IF GVL.Error_code=0 AND GVL.eAzErrorcode = 0 AND NOT GVL.bAzCtrlBit7  AND NOT tr AND NOT bfin1 AND NOT bfin2 THEN
	IF GVL.bLocalCtrl=FALSE THEN //远控
		IF sCtrl.iMode <> 1 THEN
			istate:=0;
			icount:=0;
		END_IF
		CASE sCtrl.iMode OF
			MODES.powerOff: // 下电
				IF NOT sStatus.Disabled THEN
					IF sStatus.Moving THEN // 运动中，先停止运动
						GVL.diAzTargetVel := 0;
						bAzCtrlBit8 := TRUE;
					ELSE
						// 写入下电控制字
						GVL.bAzCtrlBit3 := FALSE;
						GVL.bAzCtrlBit0 := FALSE;
						GVL.bAzCtrlBit1 := FALSE;
						GVL.bAzCtrlBit2 := FALSE;
					END_IF
				END_IF
				
				vpid1(rKpbase:=1, rKibase:=0.01, rKpMax:=1, rKiMax:=0.01, rVelThreshold:=10,rTarget:=sCtrl.rPIDCmdPos,rFeedback:=rRealPos,rPosLimPositive:=sCtrl.rSoft_limit_Postive,
							rPosLimNegitive:=sCtrl.rSoft_limit_Negative,
								bPIDEnable:=sCtrl.bPIDEnable,rVelLim:=sCtrl.rVel_Limit,rKpScale:=0.02,rKiScale:=0.005,rElPos:=GVL.rFctPosReal_1-90,
								iThrehold:=sCtrl.rPIDThre,rPIDOutDir=>sCtrl.rPIDCmdVel);
			MODES.powerOn:  // 上电
				IF sStatus.Disabled THEN
					// 目标速度清零
					GVL.diAzTargetVel := 0;
					IF GVL.siAzMode <> 3 THEN // 上电时模式默认为3，速度模式
						GVL.siAzMode := 3;
					END_IF
					IF siAzMode = 3 THEN
						CASE istate OF
							0:
								GVL.bAzCtrlBit1 := TRUE;
								GVL.bAzCtrlBit2 := TRUE;
								icount := icount + 1;
								IF icount = 20 THEN
									icount:=0;
									istate:=1;
								END_IF
							1:
								GVL.bAzCtrlBit0 := TRUE;
								icount := icount + 1;
								IF icount = 20 THEN
									icount:=0;
									istate:=2;
								END_IF
							2:
								GVL.bAzCtrlBit3 := TRUE;
						END_CASE
					END_IF
				ELSE
					IF sStatus.Moving THEN
						GVL.diAzTargetVel := 0;
						bAzCtrlBit8 := TRUE;
					ELSE
						bAzCtrlBit8 := FALSE;
					END_IF
				END_IF
			MODES.positionMode: // 远控指向模式
				IF NOT sStatus.Disabled THEN
					IF sCtrl.bStartAutoTrack THEN
						//自跟踪模式下，由误差电压直接驱动
						VelPID_1(rTarget:=sCtrl.rChanU + rRealPos,
								rFeedback:=rRealPos,
								rPosLimPositive:=sCtrl.rSoft_limit_Postive,
								rPosLimNegative:=sCtrl.rSoft_limit_Negative,
								rVelLim:=sCtrl.rVel_Limit,
								rKp:=1,//自跟踪PI系数3,0.02
								rKi:=0,
								rKd:=0,
								bPIDEnable:=sCtrl.bPIDEnable,
								iThreshold:= -1,
								rPIDOutput=>sCtrl.rPIDCmdVel);							
					ELSE
						//PID计算速度指令
						VelPID_1(rTarget:=sCtrl.rPosCmd,
							rFeedback:=rRealPos,
							rVelLim:=sCtrl.Pos_Vel,
							rPosLimPositive:=sCtrl.rSoft_limit_Postive,
							rPosLimNegative:=sCtrl.rSoft_limit_Negative,
							rKp:=0.6,//程引PI系数低带：1,0.002  高带：3,0.02
							rKi:=0,
							rKd:=0,
							bPIDEnable:=sCtrl.bPIDEnable,
							iThreshold:=sCtrl.rPIDThre,
							rPIDOutput=>sCtrl.rPIDCmdVel);
					END_IF
					GVL.diAzTargetVel := REAL_TO_DINT(sCtrl.rPIDCmdVel * 524288 / 360);
					GVL.diAzTargetAcc := REAL_TO_UDINT(12 * 524288 / 360);   //加速度
					GVL.diAzTargetDec := REAL_TO_UDINT(12 * 524288 / 360);   //减速度
				END_IF
			MODES.velocityMode://手控速度模式-远控模式
				IF NOT sStatus.Disabled THEN
					IF ABS(sCtrl.rVelCmd) <= sCtrl.rVel_Limit THEN
						GVL.diAzTargetVel := REAL_TO_DINT(sCtrl.rVelCmd * 524288 / 360);
					ELSIF sCtrl.rVelCmd > sCtrl.rVel_Limit THEN
						GVL.diAzTargetVel := REAL_TO_DINT(sCtrl.rVel_Limit * 524288 / 360);
					ELSE
						GVL.diAzTargetVel := REAL_TO_DINT(-sCtrl.rVel_Limit * 524288 / 360);
					END_IF
					GVL.diAzTargetAcc := REAL_TO_UDINT(sCtrl.rAcceleration * 524288 / 360);   //加速度
					GVL.diAzTargetDec := REAL_TO_UDINT(sCtrl.rDeceleration * 524288 / 360);   //减速度
				END_IF
			MODES.programBootMode://PID速度模式-正常模式 程引
				IF NOT sStatus.Disabled THEN
					IF sCtrl.bStartAutoTrack THEN
						(*
						//自跟踪模式下，由误差电压直接驱动
						VelPID_3(rTarget:=sCtrl.rChanU + rRealPos,
								rFeedback:=rRealPos,
								rPosLimPositive:=sCtrl.rSoft_limit_Postive,
								rPosLimNegative:=sCtrl.rSoft_limit_Negative,
								rVelLim:=sCtrl.rVel_Limit,
								rKp:=sCtrl.rP_AutoTrack,//自跟踪PI系数3,0.02
								rKi:=sCtrl.rI_AutoTrack,
								rKd:=sCtrl.rD,
								bPIDEnable:=sCtrl.bPIDEnable,
								iThreshold:= -1,
								rPIDOutput=>sCtrl.rPIDCmdVel);
								*)
						vpid1(rKpbase:=Persistentvars.rAzKpBase, rKibase:=Persistentvars.rAzKiBase, rKpMax:=Persistentvars.rAzKpMax, rKiMax:=Persistentvars.rAzKiMax, rVelThreshold:=Persistentvars.rAzThre,rTarget:=sCtrl.rPIDCmdPos,rFeedback:=rRealPos,rPosLimPositive:=sCtrl.rSoft_limit_Postive,
							rPosLimNegitive:=sCtrl.rSoft_limit_Negative,
								bPIDEnable:=sCtrl.bPIDEnable,rVelLim:=sCtrl.rVel_Limit,rKpScale:=Persistentvars.rAzKpscale,rKiScale:=Persistentvars.rAzKiscale,rElPos:=GVL.rFctPosReal_1-90,
								iThrehold:=sCtrl.rPIDThre,rPIDOutDir=>sCtrl.rPIDCmdVel);							
					ELSE
						//PID计算速度指令
						(*
						VelPID_3(rTarget:=sCtrl.rPIDCmdPos,
							rFeedback:=rRealPos,
							rVelLim:=sCtrl.rVel_Limit,
							rPosLimPositive:=sCtrl.rSoft_limit_Postive,
							rPosLimNegative:=sCtrl.rSoft_limit_Negative,
							rKp:=sCtrl.rP,//程引PI系数地带：1,0.002  高带：3,0.02
							rKi:=sCtrl.rI,
							rKd:=sCtrl.rD,
							bPIDEnable:=sCtrl.bPIDEnable,
							iThreshold:=sCtrl.rPIDThre,
							rPIDOutput=>);
							*)
						vpid1(rKpbase:=Persistentvars.rAzKpBase, rKibase:=Persistentvars.rAzKiBase, rKpMax:=Persistentvars.rAzKpMax, rKiMax:=Persistentvars.rAzKiMax, rVelThreshold:=Persistentvars.rAzThre,rTarget:=sCtrl.rPIDCmdPos,rFeedback:=rRealPos,rPosLimPositive:=sCtrl.rSoft_limit_Postive,
							rPosLimNegitive:=sCtrl.rSoft_limit_Negative,
								bPIDEnable:=sCtrl.bPIDEnable,rVelLim:=sCtrl.rVel_Limit,rKpScale:=Persistentvars.rAzKpscale,rKiScale:=Persistentvars.rAzKiscale,rElPos:=GVL.rFctPosReal_1-90,
								iThrehold:=sCtrl.rPIDThre,rPIDOutDir=>sCtrl.rPIDCmdVel);
						
					END_IF
					GVL.diAzTargetVel := REAL_TO_DINT(sCtrl.rPIDCmdVel * 524288 / 360);
					GVL.diAzTargetAcc := REAL_TO_UDINT(sCtrl.rAcceleration * 524288 / 360);   //加速度
					GVL.diAzTargetDec := REAL_TO_UDINT(sCtrl.rDeceleration * 524288 / 360);   //减速度
				END_IF
			MODES.reset://重置
				IF NOT sStatus.Disabled THEN
					IF sStatus.Moving THEN
						GVL.diAzTargetVel := 0;
						bAzCtrlBit8 := TRUE;
					ELSE
						bAzCtrlBit8 := FALSE;
					END_IF
				END_IF
			MODES.halt://待机
				IF NOT sStatus.Disabled THEN
					IF sStatus.Moving THEN
						GVL.diAzTargetVel := 0;
						bAzCtrlBit8 := TRUE;
					ELSE
						bAzCtrlBit8 := FALSE;
					END_IF
				END_IF
			
		END_CASE
	ELSE // 本控
		IF sLocal.iMode <> 1 THEN
			istate:=0;
			icount:=0;
		END_IF
		CASE sLocal.iMode OF
			MODES.powerOff: // 下电
				IF NOT sStatus.Disabled THEN
					IF sStatus.Moving THEN // 运动中，先停止运动
						GVL.diAzTargetVel := 0;
						bAzCtrlBit8 := TRUE;
					ELSE
						// 写入下电控制字
						GVL.bAzCtrlBit3 := FALSE;
						GVL.bAzCtrlBit0 := FALSE;
						GVL.bAzCtrlBit1 := FALSE;
						GVL.bAzCtrlBit2 := FALSE;
					END_IF
				END_IF
			MODES.powerOn:  // 上电
				IF sStatus.Disabled THEN
					// 目标速度清零
					GVL.diAzTargetVel := 0;
					IF GVL.siAzMode <> 3 THEN // 上电时模式默认为3，速度模式
						GVL.siAzMode := 3;
					END_IF
					IF siAzMode = 3 THEN
						CASE istate OF
							0:
								GVL.bAzCtrlBit1 := TRUE;
								GVL.bAzCtrlBit2 := TRUE;
								icount := icount + 1;
								IF icount = 20 THEN
									icount:=0;
									istate:=1;
								END_IF
							1:
								GVL.bAzCtrlBit0 := TRUE;
								icount := icount + 1;
								IF icount = 20 THEN
									icount:=0;
									istate:=2;
								END_IF
							2:
								GVL.bAzCtrlBit3 := TRUE;
						END_CASE
					END_IF
				ELSE
					IF sStatus.Moving THEN
						GVL.diAzTargetVel := 0;
						bAzCtrlBit8 := TRUE;
					ELSE
						bAzCtrlBit8 := FALSE;
					END_IF
				END_IF
			MODES.velocityMode://手控速度模式-本控模式
				IF NOT sStatus.Disabled THEN
					IF ABS(sLocal.rVelCmd) <= sLocal.rVel_Limit THEN
						GVL.diAzTargetVel := REAL_TO_DINT(sLocal.rVelCmd * 524288 / 360);
					ELSIF sLocal.rVelCmd > sLocal.rVel_Limit THEN
						GVL.diAzTargetVel := REAL_TO_DINT(sLocal.rVel_Limit * 524288 / 360);
					ELSE
						GVL.diAzTargetVel := REAL_TO_DINT(-sLocal.rVel_Limit * 524288 / 360);
					END_IF
					GVL.diAzTargetAcc := REAL_TO_UDINT(sLocal.rAcceleration * 524288 / 360);   //加速度
					GVL.diAzTargetDec := REAL_TO_UDINT(sLocal.rDeceleration * 524288 / 360);   //减速度
				END_IF
			MODES.programBootMode://本控位置模式
				IF NOT sStatus.Disabled THEN
					IF NOT sLocal.bPIDEnable THEN
						GVL.diAzTargetVel := 0;							
					ELSE
						IF NOT slocal.bStartAutoTrack THEN
							//PID计算速度指令
							 VelPID_2(rTarget:=sLocal.rPosCmd,
									 rFeedback:=rRealPos,
									 rPosLimPositive:=sLocal.rSoft_limit_Postive,//软限位
									 rPosLimNegative:=sLocal.rSoft_limit_Negative,
									 rKp:=0.6,
									 rKi:=0,
									 rKd:=0,
									 iThreshold:=sLocal.rPIDThre,
									 bPIDEnable:=sLocal.bPIDEnable,
									 rVelLim:=sLocal.Pos_Vel,
									 rPIDOutput=>sLocal.rPIDCmdVel);//普通PID
						ELSE
							//PID计算速度指令
							 VelPID_2(rTarget:=sLocal.rChanU + rRealPos,
								rFeedback:=rRealPos,
								rPosLimPositive:=sLocal.rSoft_limit_Postive,
								rPosLimNegative:=sLocal.rSoft_limit_Negative,
								rVelLim:=sLocal.rVel_Limit,
								rKp:=1,//自跟踪PI系数3,0.02
								rKi:=0,
								rKd:=0,
								bPIDEnable:=sLocal.bPIDEnable,
								iThreshold:= -1,
								rPIDOutput=>sLocal.rPIDCmdVel);//普通PID
						END_IF
						
					END_IF
					GVL.diAzTargetVel := REAL_TO_DINT(sLocal.rPIDCmdVel * 524288 / 360);
					GVL.diAzTargetAcc := REAL_TO_UDINT(12 * 524288 / 360);   //加速度
					GVL.diAzTargetDec := REAL_TO_UDINT(12 * 524288 / 360);   //减速度
				END_IF
			MODES.reset://重置
			// 是否需要
			MODES.halt://待机
				IF NOT sStatus.Disabled THEN
					IF sStatus.Moving THEN
						GVL.diAzTargetVel := 0;
						bAzCtrlBit8 := TRUE;
					ELSE
						bAzCtrlBit8 := FALSE;
					END_IF
				END_IF
			
		END_CASE
	END_IF
ELSIF GVL.Error_code<>0 AND GVL.eAzErrorcode = 0 AND NOT GVL.bAzCtrlBit7  AND NOT tr AND NOT bfin1 AND NOT bfin2 THEN
	// 出现错误，轴停止运动
	GVL.diAzTargetVel := 0;
	bAzCtrlBit8 := TRUE;
	TON_0(IN:=bAzCtrlBit8,PT:=T#1S,Q=>,ET=>);//判断stop0执行是否超时,若超时强制下电（手动复位）
	IF TON_0.Q THEN
		bTick:=TRUE;
	END_IF
	IF bTick AND sStatus.Moving THEN // 超时强制下电
		// 写入下电控制字
		GVL.bAzCtrlBit3 := FALSE;
		GVL.bAzCtrlBit0 := FALSE;
		GVL.bAzCtrlBit1 := FALSE;
		GVL.bAzCtrlBit2 := FALSE;
	END_IF
END_IF

END_FUNCTION_BLOCK

// Device/Application/PID
FUNCTION_BLOCK PID
VAR_INPUT
    rTarget : REAL;       (* 设定值 *)
    rFeedback : REAL;       (* 反馈值 *)
	rPosLimPositive:LREAL;//位置正限位
	rPosLimNegative:LREAL;//位置反限位
	rKp:REAL;     //比例增益
	rKi:REAL;     //积分增益
	rKd:REAL;     //微分增益
	iThreshold:INT;//积分项开启的位置阈值
	bPIDEnable:BOOL:=TRUE;//PID使能
	rVelLim:LREAL;//速度限制
END_VAR
VAR_OUTPUT
    rPIDOutput : LREAL:=0;         //带方向的输出速度
	rPIDtrace : LREAL:=0;         //带方向的输出速度
END_VAR
VAR
	//rPIDOutPut: REAL:=0.0;
	rLastError: LREAL:=0.0;(*上一次误差*)
	rErrorNow:LREAL:=0.0;(*当前误差*)
    rIntegralNew : LREAL := 0.0; (* 积分项 *)
    rDerivativeNew : LREAL := 0.0; (* 微分项 *)
	rDelta: LREAL;(*增量*)
	rProportionNew: LREAL;
	
	//iAzPIDEnable: INT;
END_VAR


IF (bPIDEnable>0) THEN //如果PID使能
	IF rTarget=rFeedback THEN
		rPIDOutput:=0;	
	ELSE
	
		rErrorNow:=rTarget-rFeedback;//计算当前误差 en
		rProportionNew:=rErrorNow;//比例项
		//积分项
		IF rFeedback>rPosLimNegative AND rFeedback<rPosLimPositive THEN //若在软限位之内，工作时开启积分项
			IF (ABS(rTarget-rFeedback)<iThreshold) THEN//位置差小于积分阈值
				rIntegralNew:= rIntegralNew+rErrorNow; //积分项
			ELSE
				rIntegralNew:=0;
			END_IF;
		ELSE //不在软限位范围内,则积分项为0
			rIntegralNew:=0;
		END_IF

		//PID输出
		rPIDOutPut:=rKp*rProportionNew+rKi*rIntegralNew;
		rPIDtrace:=rKp*rProportionNew+rKi*rIntegralNew;


		//PID限速
		
			IF rPIDOutput<(-rVelLim) THEN
				rPIDOutput:=-rVelLim;
			ELSIF rPIDOutput>rVelLim THEN
				rPIDOutput:=rVelLim;
			END_IF
		
		
		IF rFeedback>rPosLimPositive AND rPIDOutput>0 THEN 
			rPIDOutput:=0;
		END_IF
		IF rFeedback<rPosLimNegative AND rPIDOutput<0 THEN
			rPIDOutput:=0;
		END_IF
		
		rLastError:=rErrorNow;//将当前误差赋值给上一次误差
		
	END_IF
ELSE//非使能清零PID各项
	rProportionNew:=0.0;
	rIntegralNew:=0.0;
	rPIDOutput:=0.0;
END_IF

END_FUNCTION_BLOCK

// Device/Application/vpid
FUNCTION_BLOCK vpid
VAR_INPUT
	rTarget : REAL;           // 设定值
    rFeedback : REAL;         // 反馈值
    rPosLimPositive : LREAL;  // 位置正限位
    rPosLimNegitive : LREAL;  // 位置反限位
    rKpBase : REAL;           // 基础比例增益
    rKiBase : REAL;           // 基础积分增益
    rVelThreshold : LREAL;     // 速度阈值，真实值除以控制频率
    rKpScale : REAL;          // 比例增益比例因子
    rKiScale : REAL;          // 积分增益比例因子
    iThrehold : INT;          // 积分项开启的位置阈值
    bPIDEnable : BOOL := TRUE;// PID使能
    rVelLim : LREAL;          // 速度限制
	rKpMax : REAL;
	rKiMax : REAL;
	rElPos : REAL;            // 俯仰角度
END_VAR

VAR_OUTPUT
    rPIDOutput : LREAL := 0;  // 控制量
	rPIDOutDir: LREAL;
END_VAR

VAR
    rLastFeedback : LREAL := 0.0; // 上一次反馈值
    rErrorNow : LREAL := 0.0;     // 当前误差
    rIntegralNew : LREAL := 0.0;  // 积分项
    rDelta : LREAL;               // 增量
    rProportionNew : LREAL;       // 比例项
    rSpeed : REAL;                // 当前速度
    rKp : REAL:=1;                   // 动态比例增益
    rKi : REAL:=0.02;                   // 动态积分增益
	rInterValueNow : LREAL := 0.0;        // 当前插值位置
	rInterValueLast : LREAL := 0.0;       // 上一次插值位置
	//rSlope :LREAL :=0; 			  //PI变化斜率
	rStep:LREAL:=0.002;                //PI变化率
	
	rKpTarget :REAL:=1;
	rKiTarget :REAL:=0.02;
	
	
END_VAR

IF (bPIDEnable) THEN // 如果PID使能
    IF rTarget = rFeedback THEN
        rPIDOutDir := 0;    
    ELSE
        rErrorNow := rTarget - rFeedback; // 计算当前误差
        rProportionNew := rErrorNow;      // 比例项
		
		IF rElPos > rVelThreshold THEN
			rKpTarget := rKpBase + rKpScale * (rElPos - rVelThreshold);
			rKiTarget := rKiBase + rKiScale * (rElPos - rVelThreshold);
		ELSE
			rKpTarget := rKpBase;
			rKiTarget := rKiBase;
		END_IF
//         rInterValueLast := rInterValueNow; // 将当前插值位置值赋值给上一次
// 		rInterValueNow := RealTimePosCal.ElCubicInter.sout*10000.0;
//         // 计算当前速度
//         // rSpeed := ABS(rFeedback - rLastFeedback);
//         rSpeed := ABS(rInterValueNow - rInterValueLast)/10000.0;
// 		
//         // 根据速度调整PI增益
//         IF rSpeed > rVelThreshold THEN
//             rKpTarget := rKpBase + rKpScale * (rSpeed - rVelThreshold);
//             rKiTarget := rKiBase + rKiScale * (rSpeed - rVelThreshold);
//         ELSE
//             rKpTarget := rKpBase;
//             rKiTarget := rKiBase;
//         END_IF
        IF rKpTarget > rKpMax THEN
			rKpTarget := rKpMax;
		END_IF
		IF rKiTarget > rKiMax THEN
			rKiTarget := rKiMax;
		END_IF
		
		IF rKp<=rKpTarget THEN
			rKp:=rKp+rStep;
		ELSE
			rKp:=rKp-rStep;
		END_IF
		IF rKi<=rKiTarget THEN
			rKi:=rKi+(rKiScale/rKpScale)*rStep;
		ELSE
			rKi:=rKi-(rKiScale/rKpScale)*rStep;
		END_IF
	END_IF
        // 积分项
        IF rFeedback > rPosLimNegitive AND rFeedback < rPosLimPositive THEN // 若在软限位之内，工作时开启积分项
            IF (ABS(rTarget - rFeedback) < iThrehold) THEN // 位置差小于积分阈值
                rIntegralNew := rIntegralNew + rErrorNow;  // 积分项
            ELSE
                rIntegralNew := rIntegralNew;  // 积分项
            END_IF;
        ELSE // 不在软限位范围内，则积分项为0
            rIntegralNew := 0;
        END_IF
        (*
        // 防止目标位置与当前位置偏差过大，导致比例项输出太大，引起震动
        IF rKp * rProportionNew > 2 THEN
            rPIDOutput := 2;
        ELSIF rKp * rProportionNew < -2 THEN
            rPIDOutput := -2;
        ELSE
            rPIDOutput := rKp * rProportionNew + rKi * rIntegralNew / 1000.0; // 由于需求积分项过小，因此积分系数在接口数据上除1000
        END_IF
        *)
		rPIDOutput := rKp * rProportionNew + rKi * rIntegralNew; // 由于需求积分项过小，因此积分系数在接口数据上除1000
        // 根据方向设置输出
        IF rPIDOutput < 0 THEN

            rPIDOutDir := rPIDOutput;
        ELSE

            rPIDOutDir := rPIDOutput;
        END_IF
        
        // PID限速
        IF (ABS(rPIDOutDir) > rVelLim) THEN
            IF rPIDOutDir < (-rVelLim) THEN
                rPIDOutDir := -rVelLim;
            ELSIF rPIDOutDir > rVelLim THEN
                rPIDOutDir := rVelLim;
            END_IF
        END_IF
        
        // 位置限位检查
        IF rFeedback > rPosLimPositive AND rPIDOutDir > 0  THEN
            rPIDOutDir := 0;
        END_IF
        IF rFeedback < rPosLimNegitive AND rPIDOutDir <= 0 THEN
            rPIDOutDir := 0;
        END_IF
        
        //rLastFeedback := rFeedback; // 将当前反馈值赋值给上一次反馈值
		//rInterValueLast := rInterValueNow; // 将当前插值位置值赋值给上一次

ELSE // 非使能清零PID各项
    rProportionNew := 0.0;
    rIntegralNew := 0.0;
    rPIDOutDir := 0.0;
    rPIDOutput := 0.0;
END_IF

END_FUNCTION_BLOCK

// Device/Application/扫描搜索/AGCMaxSearch_PB_1
FUNCTION_BLOCK AGCMaxSearch_PB_1 //双轴静止星步进跟踪使用的代码
VAR_INPUT
	bstart:BOOL;//模块开始标识
	rAGCNow:REAL;//当前AGC值
	btrig:BOOL;//触发一次
	rStepBiasNow:REAL;//当前拉偏量 //用来判断此次搜索是否有效
	bAutoTracking:BOOL;// 自跟踪标识
	bStop:BOOL;//满足ua ue很小
	
	rCurrentPos:REAL;//当前位置
	rInterPos:REAL;//插值位置
	//rOutStepBias:REAL;//外部拉偏量
END_VAR
VAR_OUTPUT
	
	rAGCMaxBias:REAL;//输出AGC最强时的拉偏量 单位为°
	bSucess :BOOL;//数出模块是否成功
	rStepBias:REAL;//步进量
END_VAR
VAR
	ton:Standard.TON;
	rTrg:Standard.R_TRIG;//初始化上升沿检测器
	rAGCInit:REAL:=0;//初始化AGC
	rPrevAGC:REAL:=0;//上一步的AGC值 单位为V
	rBiasInit:REAL;//初始化拉偏量
	
	iCountStep:INT:=0;//计步数
	toN1: Standard.Ton;//计时器 定时触发上升沿 
	
	rDirection: INT:=1;
	rSearchNextStepTarget:REAL;//搜索当前目标位置 单位为°
	rStep:REAL:=0.0003;//步进值
	rSensitivity:REAL:=0.05;//反向灵敏度
	iCountStopMax:INT:=20;//停止计数上限
	
	rLastDirection:INT;//上一次方向，判断是否换向
	iCountDirChange:INT;//换向标识
	rAGCMaxPos:REAL;//信号最强位置
	
	rAGCLastrecord: REAL;
	iStatus: INT;
	iCountStop1:INT;//第一阶段停止标识 (正向)
	iCountStop2:INT;//(反向)
	
	rAGCMaxValue: REAL;//AGC最大值
	
	//新加的
	iCountSearchRight:INT;//搜索方向正确，提前结束标识
	
	bSearchRight:BOOL;//搜索正确标识
	//模块指行完成标识
	iCountBlockEnd:INT;//用来计数确认已达到最强位置
	iCountBlockEndMax:INT:=500;//到位计数上限
END_VAR


rTrg(CLK:=bstart,Q=>);

IF rTrg.Q THEN
	rAGCInit:=rAGCNow;
	rAGCMaxValue:=rAGCNow;
	//rBiasInit:=rCurrentPos-rInterPos;//获取启动时的拉偏量
END_IF

IF bstart THEN
	//搜索换向两次
	IF iCountDirChange=2 THEN
		rSearchNextStepTarget:=rAGCMaxBias;
		IF rStepBias< rSearchNextStepTarget THEN 
			rStepBias:=rStepBias+rStep;
		ELSIF rStepBias> rSearchNextStepTarget THEN
			rStepBias:=rStepBias-rStep;
		ELSE
			rStepBias:=rStepBias;
		END_IF
		
		IF ABS((rInterPos+rStepBias)-rCurrentPos)<0.002 THEN //若位置达到最强位置，则输出成功 //可能只是路过这里,需要持续
			//需要判断稳定
			iCountBlockEnd:=iCountBlockEnd+1;
		ELSE
			iCountBlockEnd:=0;
		END_IF
		IF iCountBlockEnd>iCountBlockEndMax THEN
			iCountBlockEnd:=iCountBlockEndMax+1;
			//用TON1秒后触发
			ton(IN:=TRUE,PT:=T#1S,Q=>,ET=>);
		END_IF
		IF ton.Q THEN
			bSucess:=TRUE;
		END_IF
	ELSE
		rStepBias:=rStepBias+rDirection*rStep;
		IF rDirection<0 THEN
			//若是向小走
			IF rCurrentPos<rInterPos THEN
				IF rAGCNow<rAGCMaxValue-rSensitivity THEN
					iCountStop1:=iCountStop1+1;
					IF iCountStop1>iCountStopMax THEN
						iCountStop1:=iCountStopMax+1;
						IF bSearchRight THEN
							iCountDirChange:=2;
						ELSE
							iCountDirChange:=iCountDirChange+1;
						END_IF
						rDirection:=rDirection*(-1);
					END_IF
				ELSE
					iCountStop1:=0;	
				END_IF
				
				//新加的 测试第一阶段搜索正确后不进行第二次搜索
				IF rAGCNow>rAGCInit+rSensitivity THEN
					iCountSearchRight:=iCountSearchRight+1;
				ELSE
					iCountSearchRight:=0;
				END_IF
				IF iCountSearchRight>200 THEN
					iCountSearchRight:=201;
					bSearchRight:=TRUE;
				END_IF
				
			END_IF
		ELSE
			//若是向正走
			IF rCurrentPos>rInterPos THEN
				IF rAGCNow<rAGCMaxValue-rSensitivity THEN
					iCountStop2:=iCountStop2+1;
					IF iCountStop2>iCountStopMax THEN
						iCountStop2:=iCountStopMax+1;
						IF bSearchRight THEN
							iCountDirChange:=2;
						ELSE
							iCountDirChange:=iCountDirChange+1;
						END_IF
						rDirection:=rDirection*(-1);
					END_IF
				ELSE
					iCountStop2:=0;	
				END_IF
				
				//新加的
				IF rAGCNow>rAGCInit+rSensitivity THEN
					iCountSearchRight:=iCountSearchRight+1;
				ELSE
					iCountSearchRight:=0;
				END_IF
				IF iCountSearchRight>200 THEN
					iCountSearchRight:=201;
					bSearchRight:=TRUE;
				END_IF
				
			END_IF
		END_IF
		(*
		IF rAGCNow<rAGCInit-0.05 THEN
			iCountStop1:=iCountStop1+1;
			IF iCountStop1>150 THEN
				iCountDirChange:=iCountDirChange+1;
				rDirection:=rDirection*(-1);
			END_IF
		ELSE
			iCountStop1:=0;	
		END_IF
		*)
		
		 // 记录最强信号的拉偏量和值
		//IF rAGCNow >= rAGCInit AND rAGCNow> rAGCMaxValue THEN
		IF  rAGCNow> rAGCMaxValue THEN
			rAGCMaxBias := rStepBias;
			rAGCMaxValue := rAGCNow;
		END_IF
	END_IF
ELSE
	rStepBias:=0;
	//清空变量
	iCountDirChange:=0;
	rAGCInit:=0;
	rAGCMaxValue:=0;
	rAGCMaxBias:=0;
	rDirection:=1;
	iCountStop1:=0;
	iCountStop2:=0;
	ton(IN:=FALSE,PT:=T#1S,Q=>,ET=>);
	//rStepBias:=0;
	rSearchNextStepTarget:=0;
	bSucess:=FALSE;
	iCountSearchRight:=0;
	bSearchRight:=FALSE;
	iCountBlockEnd:=0;
END_IF


(*
IF rStepBias< rSearchNextStepTarget THEN 
	rStepBias:=rStepBias+rStep;
ELSIF rStepBias> rSearchNextStepTarget THEN
	rStepBias:=rStepBias-rStep;
ELSE
	rStepBias:=rStepBias;
END_IF*)

END_FUNCTION_BLOCK

// Device/Application/El_ctrl_1
PROGRAM El_ctrl_1
VAR
    Axis1_Ctrl : El_Ctrl_FB;
    bRemote2LocalStop : BOOL;
    bLocal2RemoteStop : BOOL;
    Error : INT;
    Axis1Limit_pos : REAL;
    Axis1Limit_Neg : REAL;
    bRTriger : Standard.R_TRIG;
    bFTriger : Standard.F_TRIG;
    Stop1_Count : INT;
    bStop_1 : BOOL;
    rPosModeStepBias : LREAL;
    rPosModeStep : LREAL := 0.005;
    rStepBiasMax : LREAL := 2;
    rStepBias : LREAL;
    rStep : LREAL := 0.002;
    rAuToStepBias : LREAL;
    rAuToStepBiasTemp : LREAL;
    rAutoStep : LREAL := 0.01;
    TbAutoTrigger : Standard.F_TRIG;
    RbAutoTrigger : Standard.R_TRIG;
    rAutoTrackingBiasMax : LREAL := 6;
    rLocalInitPosModeSpeed : REAL;
    rRemoteInitPosModeSpeed : REAL;
    iCountOffAuto : INT;
    iCasePBAutoTrack : INT := 2;
    rKAuToStepBias : LREAL := 0.45; // 对齐2.4
    agcmaxsearch_tb : AGCMaxSearch_PB_1;
    rSearchNextStepTarget_tb : REAL;
    agcmaxsearch_pb : AGCMaxSearch_PB_1;
    rElthreshold : REAL := 4.2;
    toN1 : Standard.Ton;
    ttime1 : TIME := T#200mS;
    bstartagcmaxsearch : BOOL;
    rSearchNextStepTarget : REAL;
    rMaxPosTest : REAL;
END_VAR

(*
//远控轴参量赋值
Axis1Remote.iMode:=Modbus_Slave.iMode_1;
Axis1Remote.rVelCmd:=Modbus_Slave.rVelcmd_1;
Axis1Remote.rPosCmd:=Modbus_Slave.rPosCmd_1;
Axis1Remote.rP:=Modbus_Slave.rP_1;
Axis1Remote.rI:=Modbus_Slave.rI_1;
Axis1Remote.rD:=Modbus_Slave.rD_1;
Axis1Remote.rPIDThre:=Modbus_Slave.rThreshold_1;
Axis1Remote.rAcceleration:=Modbus_Slave.rAcceleration_1;
Axis1Remote.rDeceleration:=Modbus_Slave.rDeceleration_1;
Axis1Remote.rVel_Limit:=Modbus_Slave.rVelLim_1;
*)
// 方位状态写入
Axis1Status.Error := GVL.bElStsBit3;
Axis1Status.ErrorID := GVL.eElErrorcode;
Axis1Status.bServo_Enable := GVL.bElStsBit0 AND GVL.bElStsBit1 AND GVL.bElStsBit2;
Axis1Status.bBrake := NOT (GVL.bElStsBit0 AND GVL.bElStsBit1 AND GVL.bElStsBit2);
Axis1Status.Disabled := NOT (GVL.bElStsBit0 AND GVL.bElStsBit1 AND GVL.bElStsBit2);
Axis1Remote.rSoft_limit_Negative:=93;Axis1Remote.rSoft_limit_Postive:=180;
Axis1Local.rSoft_limit_Negative:=93;Axis1Local.rSoft_limit_Postive:=180;

//速度的写入
rFctVelReal_1:=DINT_TO_REAL(diElActVel)/524288.0*360.0;
//位置的写入，方位0对应编码器0，所以实际方位是：-1*编码器值
//rFctPosReal_1:=DINT_TO_REAL(diElActPos)/524288.0*360.0 + 5.339;
rFctPosReal_1:=DINT_TO_REAL(diElActPos)/524288.0*360.0 + modbus_slave.lrElOffset;
//软限位控制
Axis1Limit_pos:=180;
Axis1Limit_Neg:=93;
IF Axis1Remote.rPosCmd>Axis1Limit_pos THEN
	Axis1Remote.rPosCmd:=180;
ELSIF Axis1Remote.rPosCmd<Axis1Limit_Neg THEN
	 Axis1Remote.rPosCmd:=93;  
END_IF

IF Axis1Local.rPosCmd>Axis1Limit_pos THEN
	Axis1Local.rPosCmd:=180;
ELSIF Axis1Local.rPosCmd<Axis1Limit_Neg THEN
	 Axis1Local.rPosCmd:=93;  
END_IF

//停止标志符号判断
IF  ABS(rFctVelReal_1)<0.035 THEN
	Stop1_Count:=Stop1_Count+1;
	IF Stop1_Count>100 THEN
		Stop1_Count:=101;
		bStop_1:=TRUE;;
	END_IF
ELSE
	Stop1_Count:=0;
	bStop_1:=FALSE;
END_IF
Axis1Status.Moving := NOT bStop_1;
//PID使能赋值
IF Axis1Remote.iMode=2 OR Axis1Remote.iMode=4 THEN
	Axis1Remote.bPIDEnable:=TRUE;
ELSE
	Axis1Remote.bPIDEnable:=FALSE;
END_IF

//本远控逻辑保护
//远控切本控逻辑保护
bRTriger(CLK:=GVL.bLocalCtrl);
bFTriger(CLK:=GVL.bLocalCtrl);

IF Axis1Status.bServo_Enable AND (bRTriger.Q ) THEN//如果速度不为0且本控发生切换，则减速停止标识为True
	bRemote2LocalStop:=TRUE;
END_IF
IF bRemote2LocalStop  THEN //若减速停止标识符为True 
	
	IF  bStop_1=TRUE THEN//且电机速度不为0 开始减速 减速完成后下使能，下使能完成后复位标识符复位
		Axis1Local.iMode:=0;
		Axis1Remote.iMode:=0;
		IF Axis1Status.bServo_Enable=FALSE THEN
			bRemote2LocalStop:=FALSE;
		END_IF
	ELSE
		Axis1Local.iMode:=7;
		Axis1Remote.iMode:=7;
	END_IF
END_IF

//本控切远控
IF Axis1Status.bServo_Enable AND (bFTriger.Q ) THEN//如果速度不为0且本控发生切换，则减速停止标识为True
	bLocal2RemoteStop:=TRUE;
END_IF
IF bLocal2RemoteStop  THEN //若减速停止标识符为True 
	
	IF  bStop_1=TRUE THEN//且电机速度不为0 开始减速 减速完成后下使能，下使能完成后复位标识符复位
		Axis1Local.iMode:=0;
		Axis1Remote.iMode:=0;
		IF Axis1Status.bServo_Enable=FALSE THEN
			bLocal2RemoteStop:=FALSE;
		END_IF
	ELSE
		Axis1Remote.iMode:=7;
		Axis1Local.iMode:=7;
	END_IF
END_IF
(*
//自跟踪
IF GVL.bStartTrack THEN
	Axis1Remote.bStartAutoTrack := TRUE;
	Axis1Remote.rChanU := AutoTrackingCal.rChanUe;
ELSE
	Axis1Remote.bStartAutoTrack := FALSE;	
	Axis1Remote.rChanU := 0;
END_IF
*)
IF Axis1Remote.iMode=2 THEN
			IF GVL.Chan1AGC>=(GVL.Chanthreshold-0.1) THEN
					agcmaxsearch_pb(bstart:=Az_ctrl_1.agcmaxsearch_tb.bSucess,rAGCNow:=GVL.Chan1AGC,btrig:=Az_ctrl_1.bstartSearchEl,
						rCurrentPos:=rFctPosReal_1,rInterPos:=Axis1Remote.rPosCmd,
				//rOutStepBias:=rStepBias,	
				rStepBiasNow:=rStepBias,bAutoTracking:=GVL.bStartTrack,bStop:=FALSE,
				rStepBias=>rSearchNextStepTarget_tb,rAGCMaxBias=>rMaxPosTest,bSucess=>);
			ELSE
				bstartagcmaxsearch:=FALSE;
				agcmaxsearch_pb(bstart:=Az_ctrl_1.agcmaxsearch_tb.bSucess,rAGCNow:=GVL.Chan1AGC,btrig:=Az_ctrl_1.bstartSearchEl,
				rCurrentPos:=rFctPosReal_1,rInterPos:=Axis1Remote.rPosCmd,
				//rOutStepBias:=rStepBias,
				rStepBiasNow:=rStepBias,bAutoTracking:=GVL.bStartTrack,bStop:=FALSE,
				rStepBias=>rSearchNextStepTarget_tb,rAGCMaxBias=>rMaxPosTest,bSucess=>);
			END_IF
		ELSIF Axis1Remote.iMode=4 AND rFctPosReal_1-90>rElthreshold  THEN
			IF GVL.Chan1AGC>=(GVL.Chanthreshold-0.1) THEN
					agcmaxsearch_pb(bstart:=Az_ctrl_1.agcmaxsearch_pb.bSucess,rAGCNow:=GVL.Chan1AGC,btrig:=Az_ctrl_1.bstartSearchEl,
						rCurrentPos:=rFctPosReal_1,rInterPos:=RealTimePosCal.rInterElPos,
				//rOutStepBias:=rStepBias,	
				rStepBiasNow:=rStepBias,bAutoTracking:=GVL.bStartTrack,bStop:=FALSE,
				rStepBias=>rSearchNextStepTarget,rAGCMaxBias=>rMaxPosTest,bSucess=>);
			ELSE
				bstartagcmaxsearch:=FALSE;
				agcmaxsearch_pb(bstart:=Az_ctrl_1.agcmaxsearch_pb.bSucess,rAGCNow:=GVL.Chan1AGC,btrig:=Az_ctrl_1.bstartSearchEl,
				rCurrentPos:=rFctPosReal_1,rInterPos:=RealTimePosCal.rInterElPos,
				//rOutStepBias:=rStepBias,
				rStepBiasNow:=rStepBias,bAutoTracking:=GVL.bStartTrack,bStop:=FALSE,
				rStepBias=>rSearchNextStepTarget,rAGCMaxBias=>rMaxPosTest,bSucess=>);
			END_IF
			//把rSearchNextStepTarget附加到AzCtrl.rPIDCmdPos上
		ELSIF Axis1Remote.iMode =0  OR Axis1Remote.iMode =7 THEN
			bstartagcmaxsearch:=FALSE;
			//rSearchNextStepTarget:=0;
			agcmaxsearch_pb(bstart:=Az_ctrl_1.agcmaxsearch_pb.bSucess,rAGCNow:=GVL.Chan1AGC,btrig:=Az_ctrl_1.bstartSearchEl,
			rCurrentPos:=rFctPosReal_1,rInterPos:=RealTimePosCal.rInterElPos,	
			//rOutStepBias:=rStepBias,
			rStepBiasNow:=rStepBias,bAutoTracking:=GVL.bStartTrack,bStop:=FALSE,
			rStepBias=>rSearchNextStepTarget,rAGCMaxBias=>rMaxPosTest,bSucess=>);
		END_IF
// 程引模式下自跟踪拉偏
IF GVL.bStartTrack AND Axis1Remote.iMode=4 THEN
	Axis1Remote.bStartAutoTrack := TRUE;
	IF rAuToStepBias > rAutoTrackingBiasMax THEN
		rAuToStepBias := rAutoTrackingBiasMax;
	ELSIF rAuToStepBias < -rAutoTrackingBiasMax THEN
		rAuToStepBias := -rAutoTrackingBiasMax;
	ELSE
		rAuToStepBiasTemp:=0.02*AutoTrackingCal.rDirSenFac*AutoTrackingCal.rChanUe;
		rAuToStepBias:=rAuToStepBias+AutoTrackingCal.rDirSenFac*rKAuToStepBias*AutoTrackingCal.rChanUe/1000.0;
	END_IF
ELSIF NOT GVL.bStartTrack AND Axis1Remote.iMode=4 THEN
	IF 	rAuToStepBias>0 THEN//关闭自跟踪后自跟踪拉偏量逐渐归0
		rAuToStepBias:=rAuToStepBias-rAutoStep;
	ELSIF rAuToStepBias<0 THEN
		rAuToStepBias:=rAuToStepBias+rAutoStep;
	ELSE
		rAuToStepBias:=0;
	END_IF
	
	IF Modbus_Slave.rBias_1>rStepBias THEN
		rStepBias:=rStepBias+rStep;
		IF rStepBias>=Modbus_Slave.rBias_1 THEN
			rStepBias:=Modbus_Slave.rBias_1;
		END_IF
	ELSIF Modbus_Slave.rBias_1<rStepBias THEN
		rStepBias:=rStepBias-rStep;
		IF rStepBias<=Modbus_Slave.rBias_1 THEN
			rStepBias:=Modbus_Slave.rBias_1;
		END_IF
	END_IF
	rAuToStepBiasTemp:=0;
ELSIF GVL.bStartTrack AND Axis1Remote.iMode=2 THEN
	Axis1Remote.bStartAutoTrack := TRUE;
	Axis1Remote.rChanU := AutoTrackingCal.rChanUe;
ELSE
	Axis1Remote.bStartAutoTrack := FALSE;	
	rAuToStepBias:=0;
	rStepBias:=0;
	rAuToStepBiasTemp:=0;
END_IF

//本控自跟踪
IF GVL.bStartLocalAutoTrack AND Axis1Local.iMode = 4 THEN
	Axis1Local.bStartAutoTrack := TRUE;
	Axis1Local.rChanU := AutoTrackingCal.rChanUeLocal;
ELSE
	Axis1Local.bStartAutoTrack := FALSE;
END_IF

//拉偏
Axis1Remote.rPIDCmdPos:=RealTimePosCal.rInterElPos+rStepBias+rAuToStepBias+rSearchNextStepTarget+SECURITYCHECK.el_out+rAuToStepBiasTemp;
//限位
IF Axis1Remote.rPIDCmdPos<93 THEN
	Axis1Remote.rPIDCmdPos:=93;
ELSIF Axis1Remote.rPIDCmdPos>180 THEN
	Axis1Remote.rPIDCmdPos:=180;
END_IF

Axis1_Ctrl(sLocal:=Axis1Local, sCtrl:=Axis1Remote, sStatus:=Axis1Status, sVisible:=Axis1Visible, rRealPos:=rFctPosReal_1, rPosLimK:=0.34);

END_PROGRAM

// Device/Application/El_Ctrl_FB
FUNCTION_BLOCK El_Ctrl_FB
VAR_INPUT
	sLocal:AxisCrtlStruct;
	sCtrl:AxisCrtlStruct;
	sStatus:AxisStatus;
	sVisible:AxisVisible;
	rRealPos:REAL;
	rPosLimK:REAL;
END_VAR
VAR_OUTPUT
	logicError:INT;
END_VAR
VAR
	VelPID_1:PID;
	VelPID_2:PID;
	VelPID_3:PID;
	vpid1:vpid;
	TON_0:TON;
	bTick:BOOL;
	tr:BOOL;
	icount1:INT := 0;
	icount2:INT := 0;
	icount3:INT := 0;
	bfin1:BOOL;
	bfin2:BOOL;
	istate:INT:=0;
	icount:INT:=0;
END_VAR

// 下电时复位控制字bit8
IF sStatus.Disabled OR (NOT sStatus.Moving) THEN
	bElCtrlBit8 := FALSE;
END_IF

//	错误复位功能
IF GVL.bError_Reset THEN
	sCtrl.iMode:=6;
	sLocal.iMode:=6;
	GVL.Error_code:=0;
END_IF
IF GVL.Error_code =0 THEN
	GVL.bError_Reset:=FALSE;
END_IF

/////////心跳报错清除/////////
IF GVL.eElErrorcode = 16#8130 AND NOT tr THEN
	GVL.bElCtrlBit7 := TRUE;
	tr:=TRUE;
	istate:=0;
	icount:=0;
	// 写入下电控制字
	GVL.bElCtrlBit3 := FALSE;
	GVL.bElCtrlBit0 := FALSE;
	GVL.bElCtrlBit1 := FALSE;
	GVL.bElCtrlBit2 := FALSE;	
END_IF
IF tr THEN
	icount1 := icount1 + 1;
END_IF
IF icount1 > 101 THEN
	icount1 := 0;
	tr := FALSE;
	GVL.bElCtrlBit7 := FALSE;
	bfin1 := TRUE;
END_IF
IF bfin1 THEN
	icount2 := icount2 + 1;
END_IF
IF icount2 > 101 THEN
	bfin1 := FALSE;
	icount2 := 0;
END_IF
//////////////////////////////

IF GVL.Error_code=0 AND GVL.eElErrorcode = 0 AND NOT GVL.bElCtrlBit7  AND NOT tr AND NOT bfin1 AND NOT bfin2 THEN
	IF GVL.bLocalCtrl=FALSE THEN //远控
		IF sCtrl.iMode <> 1 THEN
			istate:=0;
			icount:=0;
		END_IF
		CASE sCtrl.iMode OF
			MODES.powerOff: // 下电
				IF NOT sStatus.Disabled THEN
					IF sStatus.Moving THEN // 运动中，先停止运动
						GVL.diElTargetVel := 0;
						bElCtrlBit8 := TRUE;
					ELSE
						// 写入下电控制字
						GVL.bElCtrlBit3 := FALSE;
						GVL.bElCtrlBit0 := FALSE;
						GVL.bElCtrlBit1 := FALSE;
						GVL.bElCtrlBit2 := FALSE;
					END_IF
				END_IF
				
				vpid1(rKpbase:=1, rKibase:=0.01, rKpMax:=1, rKiMax:=0.01, rVelThreshold:=10,rTarget:=sCtrl.rPIDCmdPos,rFeedback:=rRealPos,rPosLimPositive:=sCtrl.rSoft_limit_Postive,
							rPosLimNegitive:=sCtrl.rSoft_limit_Negative,
								bPIDEnable:=sCtrl.bPIDEnable,rVelLim:=sCtrl.rVel_Limit,rKpScale:=0.02,rKiScale:=0.005,rElPos:=GVL.rFctPosReal_1-90,
								iThrehold:=sCtrl.rPIDThre,rPIDOutDir=>sCtrl.rPIDCmdVel);
			MODES.powerOn:  // 上电
				IF sStatus.Disabled THEN
					// 目标速度清零
					GVL.diElTargetVel := 0;
					IF GVL.siElMode <> 3 THEN // 上电时模式默认为3，速度模式
						GVL.siElMode := 3;
					END_IF
					IF siElMode = 3 THEN
						CASE istate OF
							0:
								GVL.bElCtrlBit1 := TRUE;
								GVL.bElCtrlBit2 := TRUE;
								icount := icount + 1;
								IF icount = 20 THEN
									icount:=0;
									istate:=1;
								END_IF
							1:
								GVL.bElCtrlBit0 := TRUE;
								icount := icount + 1;
								IF icount = 20 THEN
									icount:=0;
									istate:=2;
								END_IF
							2:
								GVL.bElCtrlBit3 := TRUE;
						END_CASE
					END_IF
				ELSE
					IF sStatus.Moving THEN
						GVL.diElTargetVel := 0;
						bElCtrlBit8 := TRUE;
					ELSE
						bElCtrlBit8 := FALSE;
					END_IF
				END_IF
			MODES.positionMode: // 远控指向模式
				IF NOT sStatus.Disabled THEN
					IF sCtrl.bStartAutoTrack THEN
						//自跟踪模式下，由误差电压直接驱动
						VelPID_1(rTarget:=sCtrl.rChanU + rRealPos,
								rFeedback:=rRealPos,
								rPosLimPositive:=sCtrl.rSoft_limit_Postive,
								rPosLimNegative:=sCtrl.rSoft_limit_Negative,
								rVelLim:=sCtrl.rVel_Limit,
								rKp:=1,//自跟踪PI系数3,0.02
								rKi:=0,
								rKd:=0,
								bPIDEnable:=sCtrl.bPIDEnable,
								iThreshold:= -1,
								rPIDOutput=>sCtrl.rPIDCmdVel);							
					ELSE
						//PID计算速度指令
						VelPID_1(rTarget:=sCtrl.rPosCmd,
							rFeedback:=rRealPos,
							rVelLim:=sCtrl.Pos_Vel,
							rPosLimPositive:=sCtrl.rSoft_limit_Postive,
							rPosLimNegative:=sCtrl.rSoft_limit_Negative,
							rKp:=0.7,//程引PI系数地带：1,0.002  高带：3,0.02
							rKi:=0,
							rKd:=0,
							bPIDEnable:=sCtrl.bPIDEnable,
							iThreshold:=sCtrl.rPIDThre,
							rPIDOutput=>sCtrl.rPIDCmdVel);
					END_IF
					GVL.diElTargetVel := REAL_TO_DINT(sCtrl.rPIDCmdVel * 524288 / 360);
					GVL.diElTargetAcc := REAL_TO_UDINT(9 * 524288 / 360);   //加速度
					GVL.diElTargetDec := REAL_TO_UDINT(9 * 524288 / 360);   //减速度
				END_IF
			MODES.velocityMode://手控速度模式-远控模式
				IF NOT sStatus.Disabled THEN
					IF ABS(sCtrl.rVelCmd) <= sCtrl.rVel_Limit THEN
						GVL.diElTargetVel := REAL_TO_DINT(sCtrl.rVelCmd * 524288 / 360);
					ELSIF sCtrl.rVelCmd > sCtrl.rVel_Limit THEN
						GVL.diElTargetVel := REAL_TO_DINT(sCtrl.rVel_Limit * 524288 / 360);
					ELSE
						GVL.diElTargetVel := REAL_TO_DINT(-sCtrl.rVel_Limit * 524288 / 360);
					END_IF
					GVL.diElTargetAcc := REAL_TO_UDINT(sCtrl.rAcceleration * 524288 / 360);   //加速度
					GVL.diElTargetDec := REAL_TO_UDINT(sCtrl.rDeceleration * 524288 / 360);   //减速度
				END_IF
			MODES.programBootMode://PID速度模式-正常模式 程引
				IF NOT sStatus.Disabled THEN
					IF sCtrl.bStartAutoTrack THEN
						(*
						//自跟踪模式下，由误差电压直接驱动
						VelPID_3(rTarget:=sCtrl.rChanU + rRealPos,
								rFeedback:=rRealPos,
								rPosLimPositive:=sCtrl.rSoft_limit_Postive,
								rPosLimNegative:=sCtrl.rSoft_limit_Negative,
								rVelLim:=sCtrl.rVel_Limit,
								rKp:=sCtrl.rP_AutoTrack,//自跟踪PI系数3,0.02
								rKi:=sCtrl.rI_AutoTrack,
								rKd:=sCtrl.rD,
								bPIDEnable:=sCtrl.bPIDEnable,
								iThreshold:= -1,
								rPIDOutput=>sCtrl.rPIDCmdVel);	
								*)
						vpid1(rKpbase:=Persistentvars.rElKpBase, rKibase:=Persistentvars.rElKiBase, rKpMax:=Persistentvars.rElKpMax, rKiMax:=Persistentvars.rElKiMax, rVelThreshold:=Persistentvars.rElThre,rTarget:=sCtrl.rPIDCmdPos,rFeedback:=rRealPos,rPosLimPositive:=sCtrl.rSoft_limit_Postive,
							rPosLimNegitive:=sCtrl.rSoft_limit_Negative,
								bPIDEnable:=sCtrl.bPIDEnable,rVelLim:=sCtrl.rVel_Limit,rKpScale:=Persistentvars.rElKpscale,rKiScale:=Persistentvars.rElKiscale,rElPos:=GVL.rFctPosReal_1-90,
								iThrehold:=sCtrl.rPIDThre,rPIDOutDir=>sCtrl.rPIDCmdVel);						
					ELSE
						//PID计算速度指令
						(*
						VelPID_3(rTarget:=sCtrl.rPIDCmdPos,
							rFeedback:=rRealPos,
							rVelLim:=sCtrl.rVel_Limit,
							rPosLimPositive:=sCtrl.rSoft_limit_Postive,
							rPosLimNegative:=sCtrl.rSoft_limit_Negative,
							rKp:=sCtrl.rP,//程引PI系数地带：1,0.002  高带：3,0.02
							rKi:=sCtrl.rI,
							rKd:=sCtrl.rD,
							bPIDEnable:=sCtrl.bPIDEnable,
							iThreshold:=sCtrl.rPIDThre,
							rPIDOutput=>);
							*)
						vpid1(rKpbase:=Persistentvars.rElKpBase, rKibase:=Persistentvars.rElKiBase, rKpMax:=Persistentvars.rElKpMax, rKiMax:=Persistentvars.rElKiMax, rVelThreshold:=Persistentvars.rElThre,rTarget:=sCtrl.rPIDCmdPos,rFeedback:=rRealPos,rPosLimPositive:=sCtrl.rSoft_limit_Postive,
							rPosLimNegitive:=sCtrl.rSoft_limit_Negative,
								bPIDEnable:=sCtrl.bPIDEnable,rVelLim:=sCtrl.rVel_Limit,rKpScale:=Persistentvars.rElKpscale,rKiScale:=Persistentvars.rElKiscale,rElPos:=GVL.rFctPosReal_1-90,
								iThrehold:=sCtrl.rPIDThre,rPIDOutDir=>sCtrl.rPIDCmdVel);
					END_IF
					GVL.diElTargetVel := REAL_TO_DINT(sCtrl.rPIDCmdVel * 524288 / 360);
					GVL.diElTargetAcc := REAL_TO_UDINT(sCtrl.rAcceleration * 524288 / 360);   //加速度
					GVL.diElTargetDec := REAL_TO_UDINT(sCtrl.rDeceleration * 524288 / 360);   //减速度
				END_IF
			MODES.reset://重置
				IF NOT sStatus.Disabled THEN
					IF sStatus.Moving THEN
						GVL.diElTargetVel := 0;
						bElCtrlBit8 := TRUE;
					ELSE
						bElCtrlBit8 := FALSE;
					END_IF
				END_IF
			MODES.halt://待机
				IF NOT sStatus.Disabled THEN
					IF sStatus.Moving THEN
						GVL.diElTargetVel := 0;
						bElCtrlBit8 := TRUE;
					ELSE
						bElCtrlBit8 := FALSE;
					END_IF
				END_IF
			
		END_CASE
	ELSE // 本控
		IF sLocal.iMode <> 1 THEN
			istate:=0;
			icount:=0;
		END_IF
		CASE sLocal.iMode OF
			MODES.powerOff: // 下电
				IF NOT sStatus.Disabled THEN
					IF sStatus.Moving THEN // 运动中，先停止运动
						GVL.diElTargetVel := 0;
						bElCtrlBit8 := TRUE;
					ELSE
						// 写入下电控制字
						GVL.bElCtrlBit3 := FALSE;
						GVL.bElCtrlBit0 := FALSE;
						GVL.bElCtrlBit1 := FALSE;
						GVL.bElCtrlBit2 := FALSE;
					END_IF
				END_IF
			MODES.powerOn:  // 上电
				IF sStatus.Disabled THEN
					// 目标速度清零
					GVL.diElTargetVel := 0;
					IF GVL.siElMode <> 3 THEN // 上电时模式默认为3，速度模式
						GVL.siElMode := 3;
					END_IF
					IF siElMode = 3 THEN
						
						
						
						CASE istate OF
							0:
								GVL.bElCtrlBit1 := TRUE;
								GVL.bElCtrlBit2 := TRUE;
								icount := icount + 1;
								IF icount = 20 THEN
									icount:=0;
									istate:=1;
								END_IF
							1:
								GVL.bElCtrlBit0 := TRUE;
								icount := icount + 1;
								IF icount = 20 THEN
									icount:=0;
									istate:=2;
								END_IF
							2:
								GVL.bElCtrlBit3 := TRUE;
						END_CASE
					END_IF
				ELSE
					IF sStatus.Moving THEN
						GVL.diElTargetVel := 0;
						bElCtrlBit8 := TRUE;
					ELSE
						bElCtrlBit8 := FALSE;
					END_IF
				END_IF
			MODES.velocityMode://手控速度模式-本控模式
				IF NOT sStatus.Disabled THEN
					IF ABS(sLocal.rVelCmd) <= sLocal.rVel_Limit THEN
						GVL.diElTargetVel := REAL_TO_DINT(sLocal.rVelCmd * 524288 / 360);
					ELSIF sLocal.rVelCmd > sLocal.rVel_Limit THEN
						GVL.diElTargetVel := REAL_TO_DINT(sLocal.rVel_Limit * 524288 / 360);
					ELSE
						GVL.diElTargetVel := REAL_TO_DINT(-sLocal.rVel_Limit * 524288 / 360);
					END_IF
					GVL.diElTargetAcc := REAL_TO_UDINT(sLocal.rAcceleration * 524288 / 360);   //加速度
					GVL.diElTargetDec := REAL_TO_UDINT(sLocal.rDeceleration * 524288 / 360);   //减速度
				END_IF
			MODES.programBootMode://本控位置模式
				IF NOT sStatus.Disabled THEN
					IF NOT sLocal.bPIDEnable THEN
						GVL.diElTargetVel := 0;							
					ELSE
						IF NOT slocal.bStartAutoTrack THEN
							//PID计算速度指令
							 VelPID_2(rTarget:=sLocal.rPosCmd,
									 rFeedback:=rRealPos,
									 rPosLimPositive:=sLocal.rSoft_limit_Postive,//软限位
									 rPosLimNegative:=sLocal.rSoft_limit_Negative,
									 rKp:=0.7,
									 rKi:=0,
									 rKd:=0,
									 iThreshold:=sLocal.rPIDThre,
									 bPIDEnable:=sLocal.bPIDEnable,
									 rVelLim:=sLocal.Pos_Vel,
									 rPIDOutput=>sLocal.rPIDCmdVel);//普通PID
						ELSE
							 VelPID_2(rTarget:=sLocal.rChanU + rRealPos,
								rFeedback:=rRealPos,
								rPosLimPositive:=sLocal.rSoft_limit_Postive,
								rPosLimNegative:=sLocal.rSoft_limit_Negative,
								rVelLim:=sLocal.rVel_Limit,
								rKp:=1,//自跟踪PI系数3,0.02
								rKi:=0,
								rKd:=0,
								bPIDEnable:=sLocal.bPIDEnable,
								iThreshold:= -1,
								rPIDOutput=>sLocal.rPIDCmdVel);
						END_IF
						
					END_IF
					GVL.diElTargetVel := REAL_TO_DINT(sLocal.rPIDCmdVel * 524288 / 360);
					GVL.diElTargetAcc := REAL_TO_UDINT(9 * 524288 / 360);   //加速度
					GVL.diElTargetDec := REAL_TO_UDINT(9 * 524288 / 360);   //减速度
				END_IF
			MODES.reset://重置
			// 是否需要
			MODES.halt://待机
				IF NOT sStatus.Disabled THEN
					IF sStatus.Moving THEN
						GVL.diElTargetVel := 0;
						bElCtrlBit8 := TRUE;
					ELSE
						bElCtrlBit8 := FALSE;
					END_IF
				END_IF
			
		END_CASE
	END_IF
ELSIF GVL.Error_code<>0 AND GVL.eElErrorcode = 0 AND NOT GVL.bElCtrlBit7  AND NOT tr AND NOT bfin1 AND NOT bfin2 THEN
	// 出现错误，轴停止运动
	GVL.diElTargetVel := 0;
	bElCtrlBit8 := TRUE;
	TON_0(IN:=bElCtrlBit8,PT:=T#1S,Q=>,ET=>);//判断stop0执行是否超时,若超时强制下电（手动复位）
	IF TON_0.Q THEN
		bTick:=TRUE;
	END_IF
	IF bTick AND sStatus.Moving THEN // 超时强制下电
		// 写入下电控制字
		GVL.bElCtrlBit3 := FALSE;
		GVL.bElCtrlBit0 := FALSE;
		GVL.bElCtrlBit1 := FALSE;
		GVL.bElCtrlBit2 := FALSE;
	END_IF
END_IF

END_FUNCTION_BLOCK

// Device/Application/READ_485
PROGRAM READ_485
VAR
	com_init:gcan.FB_Com_Init;      		//gcan.FB_Com_Init为串口初始化功能块，可设定串口端口号，串口波特率等参数
	com_read:gcan.FB_Com_Read ;				//gcan.FB_Com_Read为串口接收功能块，用于通过接收串口发送给PLC的数据
	com_write:gcan.FB_Com_Write ;			//gcan.FB_Com_Write为串口发送功能块，用于发送串口数据
	m_uiError:UINT;							//用于承接功能块中报错引脚错误信息的变量
	m_out:BOOL;								//用于承接功能块中完成标志引脚数据的变量
	isFirst:BOOL:=TRUE;						//用于判断初始化只执行一次的逻辑
	mPort:BYTE;								//程序中用作设定串口端口号
	recSize:UINT;							//接收数据长度，单位：字节
	recBuf:ARRAY[0..19] OF BYTE;			//用于存放接收到的串口数据的数组
	recData:ARRAY[0..8] OF BYTE;			//用于存放整帧数据
	wAGC:WORD; // agc，电平值
	iUa:INT; // 方位误差电压，mV
	iUe:INT; // 俯仰误差电压，mV
	iChan1DataLen: UINT;
	chan1_i: INT;
	chan1_j: INT;
	Word2Bit1:Word2Bit;
	Word2Bit2:Word2Bit;
	Word2Bit3:Word2Bit;
	rUagcTemp:REAL;
	rUaTemp:REAL;
	rUeTemp:REAL;
	btest:BOOL;
	btest2:BOOL;
	
	rSData:REAL;
	rQData:REAL;
	Dword2Bit1:Dword2Bit;
	Dword2Bit2:Dword2Bit;
	Chan1EB_N0: REAL;
	bEBN0Lock:BOOL;
	icount0:INT;
END_VAR

mPort:=2;								//串口端口号设定，GCAN-PLC-400、GCAN-PLC-510、GCAN-PLC-511，1为232，2为485
										//GCAN-PLC-324、GCAN-PLC-326，1为第一路485，2为第2路485
IF isFirst THEN
	com_init(							//串口初始化功能块
	EN_IN:=TRUE,						//串口初始化功能块使能
	xEnable:=TRUE,						//串口功能使能
	bPort:=mPort,						//串口端口号设定
	uiBaudrate:=19200,					//串口波特率设定
	bParity:=0,							//串口奇偶校验设定，0为无校验，1为奇校验，2为偶检验
	bDatabits:=8,						//数据位设定
	bStopbits:=1,						//停止位设定
	EN_OUT=>m_out,						//串口初始化功能块执行完成标志位
	uiError=>m_uiError);				//串口初始化功能块执行错误信息
	isfirst:=FALSE;						//执行一次初始化后关闭IF的条件使其之后进入ELSE程序段运行

ELSE
	com_read(						//串口读取功能块
	EN_in:=TRUE,					//读取功能块使能，为TRUE执行读取
	bPort:=mPort,					//串口端口号设定
	p_brxdata:=ADR(recBuf),			//读取到的串口数据引脚为指针类型，使用ADR()指向自建数组将数据存放到数组中
	uiMaxsize:=20,					//设定最大读取长度
	EN_out=>m_out,					//串口读取功能块执行完成标志位******功能块执行完成不代表接收完成********
	uiRecSize=>recSize,				//串口接收数据长度，单位：字节，大于0时说明接收到数据可用于判断是否接收
	uierror=>m_uierror);			//串口读取功能块执行错误信息
	
	//GVL.Chan1Lock := BYTE_TO_BOOL(recBuf[1]);
	IF recBuf[1] = 1 AND GVL.Chan1AGC >= GVL.Chanthreshold THEN
		GVL.Chan1Lock := TRUE;
	ELSE
		GVL.Chan1Lock := FALSE;
	END_IF
	Word2Bit1.Apart_Byte[1] := recBuf[2];
	Word2Bit1.Apart_Byte[2] := recBuf[3];
	wAGC:=Word2Bit1.Apart_Word;
	
	Word2Bit2.Apart_Byte[1] := recBuf[4];
	Word2Bit2.Apart_Byte[2] := recBuf[5];
	iUa:=Word2Bit2.Apart_INT;
	
	Word2Bit3.Apart_Byte[1] := recBuf[6];
	Word2Bit3.Apart_Byte[2] := recBuf[7];
	iUe:=Word2Bit3.Apart_INT;
	IF ABS(INT_TO_REAL(iUa) * 5 / 2048) <= 5 AND ABS(INT_TO_REAL(iUe) * 5 / 2048) <= 5 AND ABS((WORD_TO_REAL(wAGC) * 5 / 76)) <=5 THEN
		GVL.Chan1Ua := INT_TO_REAL(iUa) * 5 / 2048;
		GVL.Chan1Ue := INT_TO_REAL(iUe) * 5 / 2048;
		GVL.Chan1AGC := 5 - (WORD_TO_REAL(wAGC) * 5 / 76);
	END_IF
	
	(*
	Dword2Bit1.Apart_Byte[4] := recBuf[8];
	Dword2Bit1.Apart_Byte[3] := recBuf[9];
	Dword2Bit1.Apart_Byte[2] := recBuf[10];
	Dword2Bit1.Apart_Byte[1] := recBuf[11];	
	
	
	Dword2Bit2.Apart_Byte[4] := recBuf[12];
	Dword2Bit2.Apart_Byte[3] := recBuf[13];
	Dword2Bit2.Apart_Byte[2] := recBuf[14];
	Dword2Bit2.Apart_Byte[1] := recBuf[15];	
	*)
	
	Dword2Bit1.Apart_Byte[3] := recBuf[8];
	Dword2Bit1.Apart_Byte[4] := recBuf[9];
	Dword2Bit1.Apart_Byte[1] := recBuf[10];
	Dword2Bit1.Apart_Byte[2] := recBuf[11];	
	
	
	Dword2Bit2.Apart_Byte[3] := recBuf[12];
	Dword2Bit2.Apart_Byte[4] := recBuf[13];
	Dword2Bit2.Apart_Byte[1] := recBuf[14];
	Dword2Bit2.Apart_Byte[2] := recBuf[15];	
	
	rQData:=DWORD_TO_REAL(Dword2Bit2.Apart_DWORD);
	rSData:=DWORD_TO_REAL(Dword2Bit1.Apart_DWORD)-rQData;
	//rSData:=INT_TO_REAL(Dword2Bit1.Apart_INT) - rQData;
	
	IF rSData<>0  AND rQData<>0  THEN
		Chan1EB_N0 := 10*LOG(ABS(rSData/rQData))+3.8;
	ELSE
		Chan1EB_N0 := 0;
	END_IF
	
	//程引、位置模式下，信噪比大于29；或上位机下发自跟踪
	IF ((GVL.Axis1Remote.iMode = 2 OR GVL.Axis1Remote.iMode = 4) AND Chan1EB_N0 >= 29)AND READ_485.recBuf[1] = 1 OR Modbus_Slave.bStartTrackAcu THEN
		icount0:=0;
		bEBN0Lock := TRUE;
	END_IF
	IF ( GVL.Axis1Remote.iMode = 4 or GVL.Axis1Remote.iMode =2 ) AND recBuf[1] = 0 THEN
		icount0:=icount0+1;
	END_IF
	IF icount0 > 400 OR (GVL.Axis1Remote.iMode = 0 OR GVL.Axis1Remote.iMode = 0) THEN
		icount0 := 401;
		bEBN0Lock := FALSE;
	END_IF
END_IF
(*
//加校验
iChan1DataLen:=recSize-1; //数据长度
	IF iChan1DataLen > 0 THEN
		FOR chan1_i:=0 TO iChan1DataLen BY 1 DO
			
			IF recBuf[chan1_i] = 16#7E THEN
				chan1_j:=0;
			END_IF
			recData[chan1_j]:=recBuf[chan1_i];
			
			chan1_j:=chan1_j+1;
			IF chan1_j=8 THEN
				Word2Bit1.Apart_Byte[1] := recData[2];
				Word2Bit1.Apart_Byte[2] := recData[3];
				wAGC:=Word2Bit1.Apart_Word;
				
				Word2Bit2.Apart_Byte[1] := recData[4];
				Word2Bit2.Apart_Byte[2] := recData[5];
				iUa:=Word2Bit2.Apart_INT;
				
				Word2Bit3.Apart_Byte[1] := recData[6];
				Word2Bit3.Apart_Byte[2] := recData[7];
				iUe:=Word2Bit3.Apart_INT;
				rUaTemp := INT_TO_REAL(iUa) * 5 / 2048;
				rUeTemp := INT_TO_REAL(iUe) * 5 / 2048;
				rUagcTemp := WORD_TO_REAL(wAGC) * 5 / 76;
				
				IF ABS(rUagcTemp)<=5 AND ABS(rUaTemp)<=5 AND ABS(rUeTemp)<=5THEN 
					GVL.Chan1Ua := rUaTemp;
					GVL.Chan1Ue := rUeTemp;
					GVL.Chan1AGC := rUagcTemp;
					IF recData[1] = 1 THEN
						GVL.Chan1Lock := TRUE;
					ELSE
						GVL.Chan1Lock := FALSE;
					END_IF
				END_IF
(* 
				IF ABS(GVL.Chan1AGC)>5 THEN GVL.Chan1AGC:=5;
				END_IF
				IF ABS(GVL.Chan1Ua)>5 THEN GVL.Chan1Ua:=0;
				END_IF
				IF ABS(GVL.Chan1Ue)>5 THEN GVL.Chan1Ue:=0;
				END_IF
				*)
				chan1_j:=0;
			END_IF
		END_FOR
	END_IF
	
	
END_IF
*)

END_PROGRAM

// Device/Application/扫描搜索/SpiralScan_1
FUNCTION_BLOCK SpiralScan_1

VAR_INPUT
    enable : BOOL;
    delta : REAL;
    n_steps : REAL;
    agc : REAL;
    locked : BOOL;
    AzError : REAL;
    ELError : REAL;
END_VAR

VAR_OUTPUT
    azimuth : REAL;
    elevation : REAL;
    done : BOOL;
    bType : BOOL;
END_VAR

VAR
    lock_count : INT;
    best_agc : REAL;
    best_az : REAL;
    best_el : REAL;
    bInit : BOOL;
    icount0 : INT;
    icount1 : INT;
    x : REAL;
    y : REAL;
    dx : REAL;
    dy : REAL;
    step_len : REAL;
    step_count : REAL;
    segment_progress : REAL;
    move_count : REAL;
    state : INT;
    az0 : REAL;
    el0 : REAL;
    az1 : REAL;
    el1 : REAL;
    segment_az_step : REAL;
    segment_el_step : REAL;
    side_repeat : REAL;
    icountInit : INT;
END_VAR

IF NOT enable THEN
    state := 0;
    azimuth := 0.0;
    elevation := 0.0;
    done := FALSE;
	lock_count := 0;
	icount0 := 0;
	segment_progress := 0.0;
	bInit := FALSE;
	best_agc := 0.0;
    best_az := 0.0;
    best_el := 0.0;
	icountInit := 0;
	bType := FALSE;
ELSE
    CASE state OF
        0:
			state := 1;
			lock_count := 0;
        1:
            IF NOT bInit THEN
				x := 0.0; y := 0.0;
				dx := 1.0; dy := 0.0;
				step_len := 1.0;
				step_count := 0.0;
				move_count := 1.0;
				side_repeat := 0.0;
				az0 := 0.0; el0 := 0.0;
				az1 := delta * x;
				el1 := delta * y;
				segment_az_step := (az1 - az0) / n_steps;
				segment_el_step := (el1 - el0) / n_steps;
				segment_progress := 0.0;
				bInit := TRUE;
			ELSE
				azimuth := az0 + segment_az_step * (segment_progress + 1.0);
				elevation := el0 + segment_el_step * (segment_progress + 1.0);
				segment_progress := segment_progress + 1.0;

				IF segment_progress >= n_steps THEN
					segment_progress := 0.0;
					az0 := az1;
					el0 := el1;
					x := x + dx;
					y := y + dy;
					move_count := move_count + 1.0;

					az1 := delta * x;
					el1 := delta * y;
					segment_az_step := (az1 - az0) / n_steps;
					segment_el_step := (el1 - el0) / n_steps;

					step_count := step_count + 1.0;
					IF step_count >= step_len THEN
						step_count := 0.0;
						IF dx = 1.0 AND dy = 0.0 THEN
							dx := 0.0; dy := 1.0;
						ELSIF dx = 0.0 AND dy = 1.0 THEN
							dx := -1.0; dy := 0.0;
						ELSIF dx = -1.0 AND dy = 0.0 THEN
							dx := 0.0; dy := -1.0;
						ELSIF dx = 0.0 AND dy = -1.0 THEN
							dx := 1.0; dy := 0.0;
						END_IF

						side_repeat := side_repeat + 1.0;
						IF side_repeat >= 2.0 THEN
							side_repeat := 0.0;
							step_len := step_len + 1.0;
						END_IF
					END_IF
				END_IF

				IF ABS(azimuth - 4 * delta) < 1E-6 AND ABS(elevation) < 1E-6 THEN
					azimuth := 0.0;
					elevation := 0.0;
					done := TRUE;
					state := 3;
				ELSE
					IF locked THEN
					   lock_count := lock_count + 1;
					ELSE
					   lock_count := 0;
					END_IF
					IF lock_count >= 10 THEN
					   azimuth := -Azerror;
            		   elevation := -elError;
					   done := TRUE;
					   state := 2;
					END_IF
				END_IF
			END_IF
        2:
            done := TRUE;
        3:
            azimuth := 0.0;
            elevation := 0.0;
            done := TRUE;
    END_CASE
	IF state = 2 THEN
		bType := TRUE;
	ELSIF state = 3 THEN
		bType := FALSE;
	END_IF
END_IF;

END_FUNCTION_BLOCK

// Device/Application/Ti_ctrl_1
PROGRAM Ti_ctrl_1
VAR
	Axis3_Ctrl:Ti_Ctrl_FB;
	bRemote2LocalStop:BOOL;
	bLocal2RemoteStop:BOOL;
	Error:INT;
	
	Axis3Limit_pos:REAL;//正软限位
	Axis3Limit_Neg:REAL;//负软限位
	
	bRTriger:Standard.R_TRIG;//本控上升沿
	bFTriger:Standard.F_TRIG;//远控下降沿
	Stop3_Count: INT;
	bStop_3: BOOL;
	
	//指向模式自跟踪
	rPosModeStepBias:LREAL;//指向模式自跟踪拉偏累计值
	rPosModeStep:LREAL:=0.005;//指向模式自跟踪步长，积分用
	rStepBiasMax:LREAL:=2;//指向模式拉偏最大值
	
	//程引拉偏
	rStepBias:LREAL;//步进拉偏累计值
// 	rStep:LREAL:=0.0002;//步长，与控制周期有关，1ms周期对应1秒内累积0.0002*1000=0.2°
// 	rStep:LREAL:=0.01;//步长，与控制周期有关，50ms周期对应1秒内累积0.01*20=0.2°
	rStep:LREAL:=0.004;//步长，与控制周期有关，20ms周期对应1秒内累积0.004*50=0.2°
		
	//自跟踪拉偏
	rAuToStepBias:LREAL;//步进拉偏累计值
// 	rAutoStep:LREAL:=0.005;//步长
	rAutoStep:LREAL:=0.01;//步长
	TbAutoTrigger:Standard.F_TRIG;//自跟踪关闭的下降沿
	RbAutoTrigger:Standard.R_TRIG;//自跟踪开启的上升沿

	rAutoTrackingBiasMax:LREAL:=300;//自跟踪拉偏最大值
	rLocalInitPosModeSpeed: REAL;
	rRemoteInitPosModeSpeed: REAL;
	iCountOffAuto: INT;
	
	iCasePBAutoTrack:INT:=2;//程序引导自跟踪切换 
// 	rKAuToStepBias:LREAL:=0.25;
	rKAuToStepBias:LREAL:=0.16;
	bVisError:BOOL; //报错可视化标识
END_VAR

IF GVL.Error_code <> 0 THEN
	bVisError := TRUE;
ELSE
	bVisError := FALSE;
END_IF
(*
//远控轴参量赋值
Axis2Remote.iMode:=Modbus_Slave.iMode_2;
Axis2Remote.rVelCmd:=Modbus_Slave.rVelcmd_2;
Axis2Remote.rPosCmd:=Modbus_Slave.rPosCmd_2;
Axis2Remote.rP:=Modbus_Slave.rP_2;
Axis2Remote.rI:=Modbus_Slave.rI_2;
Axis2Remote.rD:=Modbus_Slave.rD_2;
Axis2Remote.rPIDThre:=Modbus_Slave.rThreshold_2;
Axis2Remote.rAcceleration:=Modbus_Slave.rAcceleration_2;
Axis2Remote.rDeceleration:=Modbus_Slave.rDeceleration_2;
Axis2Remote.rVel_Limit:=Modbus_Slave.rVelLim_2;
*)
// 倾斜轴状态写入
Axis3Status.Error := GVL.bTiStsBit3;
Axis3Status.ErrorID := GVL.eTiErrorcode;
Axis3Status.bServo_Enable := GVL.bTiStsBit0 AND GVL.bTiStsBit1 AND GVL.bTiStsBit2;
Axis3Status.bBrake := NOT (GVL.bTiStsBit0 AND GVL.bTiStsBit1 AND GVL.bTiStsBit2);
Axis3Status.Disabled := NOT (GVL.bTiStsBit0 AND GVL.bTiStsBit1 AND GVL.bTiStsBit2);
Axis3Remote.rSoft_limit_Negative:=-190;Axis3Remote.rSoft_limit_Postive:=190;
Axis3Local.rSoft_limit_Negative:=-190;Axis3Local.rSoft_limit_Postive:=190;

//速度的写入
rFctVelReal_3:=DINT_TO_REAL(diTiActVel)/524288.0*360.0;
//位置的写入，方位0对应编码器0，所以实际方位是：-1*编码器值
//rFctPosReal_3:=DINT_TO_REAL(diTiActPos)/524288.0*360.0-11.413-0.08;
rFctPosReal_3:=DINT_TO_REAL(diTiActPos)/524288.0*360.0;
//软限位控制
Axis3Limit_pos:=190;
Axis3Limit_Neg:=-190;
IF Axis3Remote.rPosCmd>Axis3Limit_pos THEN
	Axis3Remote.rPosCmd:=190;
ELSIF Axis3Remote.rPosCmd<Axis3Limit_Neg THEN
	 Axis3Remote.rPosCmd:=-190;  
END_IF

IF Axis3Local.rPosCmd>Axis3Limit_pos THEN
	Axis2Local.rPosCmd:=190;
ELSIF Axis3Local.rPosCmd<Axis3Limit_Neg THEN
	 Axis3Local.rPosCmd:=-190;  
END_IF

//停止标志符号判断
IF  ABS(rFctVelReal_3)<0.035 THEN
	Stop3_Count:=Stop3_Count+1;
	IF Stop3_Count>100 THEN
		Stop3_Count:=101;
		bStop_3:=TRUE;;
	END_IF
ELSE
	Stop3_Count:=0;
	bStop_3:=FALSE;
END_IF
Axis3Status.Moving := NOT bStop_3;
//PID使能赋值
IF Axis3Remote.iMode=2 OR Axis3Remote.iMode=4 THEN
	Axis3Remote.bPIDEnable:=TRUE;
ELSE
	Axis3Remote.bPIDEnable:=FALSE;
END_IF

//本远控逻辑保护
//远控切本控逻辑保护
bRTriger(CLK:=GVL.bLocalCtrl);
bFTriger(CLK:=GVL.bLocalCtrl);

IF Axis3Status.bServo_Enable AND (bRTriger.Q ) THEN//如果速度不为0且本控发生切换，则减速停止标识为True
	bRemote2LocalStop:=TRUE;
END_IF
IF bRemote2LocalStop  THEN //若减速停止标识符为True 
	
	IF  bStop_3=TRUE THEN//且电机速度不为0 开始减速 减速完成后下使能，下使能完成后复位标识符复位
		Axis3Local.iMode:=0;
		Axis3Remote.iMode:=0;
		IF Axis3Status.bServo_Enable=FALSE THEN
			bRemote2LocalStop:=FALSE;
		END_IF
	ELSE
		Axis3Remote.iMode:=7;
	END_IF
END_IF

//本控切远控
IF Axis3Status.bServo_Enable AND (bFTriger.Q ) THEN//如果速度不为0且本控发生切换，则减速停止标识为True
	bLocal2RemoteStop:=TRUE;
END_IF
IF bLocal2RemoteStop  THEN //若减速停止标识符为True 
	
	IF  bStop_3=TRUE THEN//且电机速度不为0 开始减速 减速完成后下使能，下使能完成后复位标识符复位
		Axis3Local.iMode:=0;
		Axis3Remote.iMode:=0;
		IF Axis3Status.bServo_Enable=FALSE THEN
			bLocal2RemoteStop:=FALSE;
		END_IF
	ELSE
		Axis3Remote.iMode:=7;
		Axis3Local.iMode:=7;
	END_IF
END_IF
(*
//自跟踪
IF GVL.bStartTrack THEN
	Axis2Remote.bStartAutoTrack := TRUE;
	Axis2Remote.rChanU := -AutoTrackingCal.rChanUa;
ELSE
	Axis2Remote.bStartAutoTrack := FALSE;	
	Axis2Remote.rChanU := 0;
END_IF
//拉偏
Axis2Remote.rPIDCmdPos:=RealTimePosCal.rInterAzPos+Modbus_Slave.rBias_2;
*)
//限位
IF Axis3Remote.rPIDCmdPos<-190 THEN
	Axis3Remote.rPIDCmdPos:=-190;
ELSIF Axis3Remote.rPIDCmdPos>190 THEN
	Axis3Remote.rPIDCmdPos:=190;
END_IF

Axis3_Ctrl(sLocal:=Axis3Local, sCtrl:=Axis3Remote, sStatus:=Axis3Status, sVisible:=Axis3Visible, rRealPos:=rFctPosReal_3, rPosLimK:=0.34);

END_PROGRAM

// Device/Application/Ti_Ctrl_FB
FUNCTION_BLOCK Ti_Ctrl_FB
VAR_INPUT
	sLocal:AxisCrtlStruct;
	sCtrl:AxisCrtlStruct;
	sStatus:AxisStatus;
	sVisible:AxisVisible;
	rRealPos:REAL;
	rPosLimK:REAL;
END_VAR
VAR_OUTPUT
	logicError:INT;
END_VAR
VAR
	VelPID_1:PID;
	VelPID_2:PID;
	TON_0:TON;
	bTick:BOOL;
	tr:BOOL;
	icount1:INT := 0;
	icount2:INT := 0;
	icount3:INT := 0;
	bfin1:BOOL;
	bfin2:BOOL;
	istate:INT:=0;
	icount:INT:=0;
END_VAR

// 下电时复位控制字bit8
IF sStatus.Disabled OR(NOT sStatus.Moving)THEN
	bTiCtrlBit8 := FALSE;
END_IF

//	错误复位功能
IF GVL.bError_Reset THEN
	sCtrl.iMode:=6;
	sLocal.iMode:=6;
	GVL.Error_code:=0;
END_IF
IF GVL.Error_code =0 THEN
	GVL.bError_Reset:=FALSE;
END_IF

/////////心跳报错清除/////////
IF GVL.eTiErrorcode = 16#8130 AND NOT tr THEN
	GVL.bTiCtrlBit7 := TRUE;
	tr:=TRUE;
	istate:=0;
	icount:=0;
	// 写入下电控制字
	GVL.bTiCtrlBit3 := FALSE;
	GVL.bTiCtrlBit0 := FALSE;
	GVL.bTiCtrlBit1 := FALSE;
	GVL.bTiCtrlBit2 := FALSE;
END_IF
IF tr THEN
	icount1 := icount1 + 1;
END_IF
IF icount1 > 101 THEN
	icount1 := 0;
	tr := FALSE;
	GVL.bTiCtrlBit7 := FALSE;
	bfin1 := TRUE;
END_IF
IF bfin1 THEN
	icount2 := icount2 + 1;
END_IF
IF icount2 > 101 THEN
	bfin1 := FALSE;
	icount2 := 0;
END_IF
/////////////////////////////

IF GVL.Error_code=0 AND GVL.eTiErrorcode = 0 AND NOT GVL.bTiCtrlBit7  AND NOT tr AND NOT bfin1 AND NOT bfin2 THEN
	IF GVL.bLocalCtrl=FALSE THEN //远控
		IF sCtrl.iMode <> 1 THEN
			istate:=0;
			icount:=0;
		END_IF
		CASE sCtrl.iMode OF
			MODES.powerOff: // 下电
				IF NOT sStatus.Disabled THEN
					IF sStatus.Moving THEN // 运动中，先停止运动
						GVL.diTiTargetVel := 0;
						bTiCtrlBit8 := TRUE;
					ELSE
						// 写入下电控制字
						GVL.bTiCtrlBit3 := FALSE;
						GVL.bTiCtrlBit0 := FALSE;
						GVL.bTiCtrlBit1 := FALSE;
						GVL.bTiCtrlBit2 := FALSE;
					END_IF
				END_IF
			MODES.powerOn:  // 上电
				IF sStatus.Disabled THEN
					// 目标速度清零
					GVL.diTiTargetVel := 0;
					IF GVL.siTiMode <> 3 THEN // 上电时模式默认为3，速度模式
						GVL.siTiMode := 3;
					END_IF
					IF siTiMode = 3 THEN
						CASE istate OF
							0:
								GVL.bTiCtrlBit1 := TRUE;
								GVL.bTiCtrlBit2 := TRUE;
								icount := icount + 1;
								IF icount = 20 THEN
									icount:=0;
									istate:=1;
								END_IF
							1:
								GVL.bTiCtrlBit0 := TRUE;
								icount := icount + 1;
								IF icount = 20 THEN
									icount:=0;
									istate:=2;
								END_IF
							2:
								GVL.bTiCtrlBit3 := TRUE;
						END_CASE
					END_IF
				ELSE
					IF sStatus.Moving THEN
						GVL.diTiTargetVel := 0;
						bTiCtrlBit8 := TRUE;
					ELSE
						bTiCtrlBit8 := FALSE;
					END_IF
				END_IF
			MODES.positionMode: // 远控指向模式
				IF NOT sStatus.Disabled THEN
					IF sCtrl.bStartAutoTrack THEN
						(*
						//自跟踪模式下，由误差电压直接驱动
						VelPID_1(rTarget:=sCtrl.rChanU + rRealPos,
								rFeedback:=rRealPos,
								rPosLimPositive:=sCtrl.rSoft_limit_Postive,
								rPosLimNegative:=sCtrl.rSoft_limit_Negative,
								rVelLim:=sCtrl.rVel_Limit,
								rKp:=sCtrl.rP_AutoTrack,//自跟踪PI系数3,0.02
								rKi:=sCtrl.rI_AutoTrack,
								rKd:=sCtrl.rD,
								bPIDEnable:=sCtrl.bPIDEnable,
								iThreshold:= -1,
								rPIDOutput=>sCtrl.rPIDCmdVel);
*)							
					ELSE
						//PID计算速度指令
						VelPID_1(rTarget:=sCtrl.rPosCmd,
							rFeedback:=rRealPos,
							rVelLim:=sCtrl.Pos_Vel,
							rPosLimPositive:=sCtrl.rSoft_limit_Postive,
							rPosLimNegative:=sCtrl.rSoft_limit_Negative,
							rKp:=0.8,//程引PI系数地带：1,0.002  高带：3,0.02
							rKi:=0,
							rKd:=0,
							bPIDEnable:=sCtrl.bPIDEnable,
							iThreshold:=sCtrl.rPIDThre,
							rPIDOutput=>sCtrl.rPIDCmdVel);
					END_IF
					GVL.diTiTargetVel := REAL_TO_DINT(sCtrl.rPIDCmdVel * 524288 / 360);
					GVL.diTiTargetAcc := REAL_TO_UDINT(10 * 524288 / 360);   //加速度
					GVL.diTiTargetDec := REAL_TO_UDINT(10 * 524288 / 360);   //减速度
				END_IF
			MODES.velocityMode://手控速度模式-远控模式
				IF NOT sStatus.Disabled THEN
					IF ABS(sCtrl.rVelCmd) <= sCtrl.rVel_Limit THEN
						GVL.diTiTargetVel := REAL_TO_DINT(sCtrl.rVelCmd * 524288 / 360);
					ELSIF sCtrl.rVelCmd > sCtrl.rVel_Limit THEN
						GVL.diTiTargetVel := REAL_TO_DINT(sCtrl.rVel_Limit * 524288 / 360);
					ELSE
						GVL.diTiTargetVel := REAL_TO_DINT(-sCtrl.rVel_Limit * 524288 / 360);
					END_IF
					GVL.diTiTargetAcc := REAL_TO_UDINT(sCtrl.rAcceleration * 524288 / 360);   //加速度
					GVL.diTiTargetDec := REAL_TO_UDINT(sCtrl.rDeceleration * 524288 / 360);   //减速度
				END_IF
			MODES.programBootMode://PID速度模式-正常模式 程引
				IF NOT sStatus.Disabled THEN
					IF sCtrl.bStartAutoTrack THEN
						//自跟踪模式下，由误差电压直接驱动
						VelPID_1(rTarget:=sCtrl.rChanU + rRealPos,
								rFeedback:=rRealPos,
								rPosLimPositive:=sCtrl.rSoft_limit_Postive,
								rPosLimNegative:=sCtrl.rSoft_limit_Negative,
								rVelLim:=sCtrl.rVel_Limit,
								rKp:=sCtrl.rP_AutoTrack,//自跟踪PI系数3,0.02
								rKi:=sCtrl.rI_AutoTrack,
								rKd:=sCtrl.rD,
								bPIDEnable:=sCtrl.bPIDEnable,
								iThreshold:= -1,
								rPIDOutput=>sCtrl.rPIDCmdVel);							
					ELSE
						//PID计算速度指令
						VelPID_1(rTarget:=sCtrl.rPIDCmdPos,
							rFeedback:=rRealPos,
							rVelLim:=sCtrl.rVel_Limit,
							rPosLimPositive:=sCtrl.rSoft_limit_Postive,
							rPosLimNegative:=sCtrl.rSoft_limit_Negative,
							rKp:=sCtrl.rP,//程引PI系数地带：1,0.002  高带：3,0.02
							rKi:=sCtrl.rI,
							rKd:=sCtrl.rD,
							bPIDEnable:=sCtrl.bPIDEnable,
							iThreshold:=sCtrl.rPIDThre,
							rPIDOutput=>sCtrl.rPIDCmdVel);
					END_IF
					GVL.diTiTargetVel := REAL_TO_DINT(sCtrl.rPIDCmdVel * 524288 / 360);
					GVL.diTiTargetAcc := REAL_TO_UDINT(sCtrl.rAcceleration * 524288 / 360);   //加速度
					GVL.diTiTargetDec := REAL_TO_UDINT(sCtrl.rDeceleration * 524288 / 360);   //减速度
				END_IF
			MODES.reset://重置
				IF NOT sStatus.Disabled THEN
					IF sStatus.Moving THEN
						GVL.diTiTargetVel := 0;
						bTiCtrlBit8 := TRUE;
					ELSE
						bTiCtrlBit8 := FALSE;
					END_IF
				END_IF
			MODES.halt://待机
				IF NOT sStatus.Disabled THEN
					IF sStatus.Moving THEN
						GVL.diTiTargetVel := 0;
						bTiCtrlBit8 := TRUE;
					ELSE
						bTiCtrlBit8 := FALSE;
					END_IF
				END_IF
			
		END_CASE
	ELSE // 本控
		IF sLocal.iMode <> 1 THEN
			istate:=0;
			icount:=0;
		END_IF
		CASE sLocal.iMode OF
			MODES.powerOff: // 下电
				IF NOT sStatus.Disabled THEN
					IF sStatus.Moving THEN // 运动中，先停止运动
						GVL.diTiTargetVel := 0;
						bTiCtrlBit8 := TRUE;
					ELSE
						// 写入下电控制字
						GVL.bTiCtrlBit3 := FALSE;
						GVL.bTiCtrlBit0 := FALSE;
						GVL.bTiCtrlBit1 := FALSE;
						GVL.bTiCtrlBit2 := FALSE;
					END_IF
				END_IF
			MODES.powerOn:  // 上电
				IF sStatus.Disabled THEN
					// 目标速度清零
					GVL.diTiTargetVel := 0;
					IF GVL.siTiMode <> 3 THEN // 上电时模式默认为3，速度模式
						GVL.siTiMode := 3;
					END_IF
					IF siTiMode = 3 THEN
						CASE istate OF
							0:
								GVL.bTiCtrlBit1 := TRUE;
								GVL.bTiCtrlBit2 := TRUE;
								icount := icount + 1;
								IF icount = 20 THEN
									icount:=0;
									istate:=1;
								END_IF
							1:
								GVL.bTiCtrlBit0 := TRUE;
								icount := icount + 1;
								IF icount = 20 THEN
									icount:=0;
									istate:=2;
								END_IF
							2:
								GVL.bTiCtrlBit3 := TRUE;
						END_CASE
					END_IF
				ELSE
					IF sStatus.Moving THEN
						GVL.diTiTargetVel := 0;
						bTiCtrlBit8 := TRUE;
					ELSE
						bTiCtrlBit8 := FALSE;
					END_IF
				END_IF
			MODES.velocityMode://手控速度模式-本控模式
				IF NOT sStatus.Disabled THEN
					IF ABS(sLocal.rVelCmd) <= sLocal.rVel_Limit THEN
						GVL.diTiTargetVel := REAL_TO_DINT(sLocal.rVelCmd * 524288 / 360);
					ELSIF sLocal.rVelCmd > sLocal.rVel_Limit THEN
						GVL.diTiTargetVel := REAL_TO_DINT(sLocal.rVel_Limit * 524288 / 360);
					ELSE
						GVL.diTiTargetVel := REAL_TO_DINT(-sLocal.rVel_Limit * 524288 / 360);
					END_IF
					GVL.diTiTargetAcc := REAL_TO_UDINT(sLocal.rAcceleration * 524288 / 360);   //加速度
					GVL.diTiTargetDec := REAL_TO_UDINT(sLocal.rDeceleration * 524288 / 360);   //减速度
				END_IF
			MODES.programBootMode://本控位置模式
				IF NOT sStatus.Disabled THEN
					IF NOT sLocal.bPIDEnable THEN
						GVL.diTiTargetVel := 0;							
					ELSE
						//PID计算速度指令
						 VelPID_2(rTarget:=sLocal.rPosCmd,
							     rFeedback:=rRealPos,
								 rPosLimPositive:=sLocal.rSoft_limit_Postive,//软限位
								 rPosLimNegative:=sLocal.rSoft_limit_Negative,
								 rKp:=sLocal.rP,
								 rKi:=sLocal.rI,
								 rKd:=sLocal.rD,
								 iThreshold:=sLocal.rPIDThre,
								 bPIDEnable:=sLocal.bPIDEnable,
								 rVelLim:=sLocal.Pos_Vel,
								 rPIDOutput=>sLocal.rPIDCmdVel);//普通PID
					END_IF
					GVL.diTiTargetVel := REAL_TO_DINT(sLocal.rPIDCmdVel * 524288 / 360);
					GVL.diTiTargetAcc := REAL_TO_UDINT(sLocal.rAcceleration * 524288 / 360);   //加速度
					GVL.diTiTargetDec := REAL_TO_UDINT(sLocal.rDeceleration * 524288 / 360);   //减速度
				END_IF
			MODES.reset://重置
			// 是否需要
			MODES.halt://待机
				IF NOT sStatus.Disabled THEN
					IF sStatus.Moving THEN
						GVL.diTiTargetVel := 0;
						bTiCtrlBit8 := TRUE;
					ELSE
						bTiCtrlBit8 := FALSE;
					END_IF
				END_IF
			
		END_CASE
	END_IF
ELSIF GVL.Error_code<>0 AND GVL.eTiErrorcode = 0 AND NOT GVL.bTiCtrlBit7  AND NOT tr AND NOT bfin1 AND NOT bfin2 THEN
	// 出现错误，轴停止运动
	GVL.diTiTargetVel := 0;
	bTiCtrlBit8 := TRUE;
	TON_0(IN:=bTiCtrlBit8,PT:=T#1S,Q=>,ET=>);//判断stop0执行是否超时,若超时强制下电（手动复位）
	IF TON_0.Q THEN
		bTick:=TRUE;
	END_IF
	IF bTick AND sStatus.Moving THEN // 超时强制下电
		// 写入下电控制字
		GVL.bTiCtrlBit3 := FALSE;
		GVL.bTiCtrlBit0 := FALSE;
		GVL.bTiCtrlBit1 := FALSE;
		GVL.bTiCtrlBit2 := FALSE;
	END_IF
END_IF

END_FUNCTION_BLOCK

// Device/Application/PLC_PRG
PROGRAM PLC_PRG
VAR
	a : DINT;
	b : REAL;
END_VAR

a := REAL_TO_DINT(b * 524288 / 360);

END_PROGRAM

// Device/Application/GPRMC
PROGRAM GPRMC
VAR
	com_init:gcan.FB_Com_Init;      		//gcan.FB_Com_Init为串口初始化功能块，可设定串口端口号，串口波特率等参数
	com_read:gcan.FB_Com_Read ;				//gcan.FB_Com_Read为串口接收功能块，用于通过接收串口发送给PLC的数据
	com_write:gcan.FB_Com_Write ;			//gcan.FB_Com_Write为串口发送功能块，用于发送串口数据
	m_uiError:UINT;							//用于承接功能块中报错引脚错误信息的变量
	m_out:BOOL;								//用于承接功能块中完成标志引脚数据的变量
	isFirst:BOOL:=TRUE;						//用于判断初始化只执行一次的逻辑
	mPort:BYTE;								//程序中用作设定串口端口号
	recSize:UINT;							//接收数据长度，单位：字节
	recBuf:ARRAY[0..100] OF BYTE;			//用于存放接收到的串口数据的数组
	sum_i:INT;
	checksum:BYTE;
	iYear: INT;
	iMonth: INT;
	iDay: INT;
	iHour: INT;
	iMinute: INT;
	iSecond: INT;
	strDateTimeNow : STRING;
	gnssTimestamp: ULINT;
	high4: BYTE;
	low4: BYTE;
END_VAR

////////////////////////////////////////////////////////////////////////////////////////
//串口接收GPRMC报文解析
//日期：2024/08/25
//版本：V1.1
/////////////////////////////////////////////////////////////////////////////////////////

mPort:=1;								//串口端口号设定，GCAN-PLC-400、GCAN-PLC-510、GCAN-PLC-511，1为232，2为485
										//GCAN-PLC-324、GCAN-PLC-326，1为第一路485，2为第2路485
IF isFirst THEN
	com_init(							//串口初始化功能块
	EN_IN:=TRUE,						//串口初始化功能块使能
	xEnable:=TRUE,						//串口功能使能
	bPort:=mPort,						//串口端口号设定
	uiBaudrate:=115200,					//串口波特率设定
	bParity:=0,							//串口奇偶校验设定，0为无校验，1为奇校验，2为偶检验
	bDatabits:=8,						//数据位设定
	bStopbits:=1,						//停止位设定
	EN_OUT=>m_out,						//串口初始化功能块执行完成标志位
	uiError=>m_uiError);				//串口初始化功能块执行错误信息
	isfirst:=FALSE;						//执行一次初始化后关闭IF的条件使其之后进入ELSE程序段运行

ELSE
	
		com_read(						//串口读取功能块
		EN_in:=TRUE,					//读取功能块使能，为TRUE执行读取
		bPort:=mPort,					//串口端口号设定
		p_brxdata:=ADR(recBuf),			//读取到的串口数据引脚为指针类型，使用ADR()指向自建数组将数据存放到数组中
		uiMaxsize:=100,					//设定最大读取长度
		EN_out=>m_out,					//串口读取功能块执行完成标志位******功能块执行完成不代表接收完成********
		uiRecSize=>recSize,				//串口接收数据长度，单位：字节，大于0时说明接收到数据可用于判断是否接收
		uierror=>m_uierror);			//串口读取功能块执行错误信息
										//从数组recBuf里取数据，解析出年、月、日、时、分、秒
		//有效判定(A)+和校验(hh),前 4bit和后 4bit的 16 进制数分别以 ASCII 码表示(0~9,A~F)，高位在前。
		IF 	recBuf[17] = 65 THEN
(*			checksum := 16#00;
			FOR sum_i:=1 TO 74 BY 1 DO
				checksum:= checksum XOR recBuf[sum_i];
			END_FOR
			high4 := (SHR(checksum, 4) AND 16#0F)+16#30;
			low4 := (checksum AND 16#0F)+16#30;
			IF recBuf[76]= high4 AND recBuf[77]= low4 THEN 
*)			IF recBuf[60] = 44 THEN // 航向角 x.x
				iYear:=BYTE_TO_INT(recBuf[65]-48)*10+BYTE_TO_INT(recBuf[66]-48)+2000;
				iMonth:=BYTE_TO_INT(recBuf[63]-48)*10+BYTE_TO_INT(recBuf[64]-48);
				iDay:=BYTE_TO_INT(recBuf[61]-48)*10+BYTE_TO_INT(recBuf[62]-48);
				iHour:=BYTE_TO_INT(recBuf[7]-48)*10+BYTE_TO_INT(recBuf[8]-48)+8;
				iMinute:=BYTE_TO_INT(recBuf[9]-48)*10+BYTE_TO_INT(recBuf[10]-48);
				iSecond:=BYTE_TO_INT(recBuf[11]-48)*10+BYTE_TO_INT(recBuf[12]-48);
			END_IF
			IF recBuf[61] = 44 THEN // 航向角 xx.x
				iYear:=BYTE_TO_INT(recBuf[66]-48)*10+BYTE_TO_INT(recBuf[67]-48)+2000;
				iMonth:=BYTE_TO_INT(recBuf[64]-48)*10+BYTE_TO_INT(recBuf[65]-48);
				iDay:=BYTE_TO_INT(recBuf[62]-48)*10+BYTE_TO_INT(recBuf[63]-48);
				iHour:=BYTE_TO_INT(recBuf[7]-48)*10+BYTE_TO_INT(recBuf[8]-48)+8;
				iMinute:=BYTE_TO_INT(recBuf[9]-48)*10+BYTE_TO_INT(recBuf[10]-48);
				iSecond:=BYTE_TO_INT(recBuf[11]-48)*10+BYTE_TO_INT(recBuf[12]-48);
			END_IF
			IF recBuf[62] = 44 THEN // 航向角 xxx.x
				iYear:=BYTE_TO_INT(recBuf[67]-48)*10+BYTE_TO_INT(recBuf[68]-48)+2000;
				iMonth:=BYTE_TO_INT(recBuf[65]-48)*10+BYTE_TO_INT(recBuf[66]-48);
				iDay:=BYTE_TO_INT(recBuf[63]-48)*10+BYTE_TO_INT(recBuf[64]-48);
				iHour:=BYTE_TO_INT(recBuf[7]-48)*10+BYTE_TO_INT(recBuf[8]-48)+8;
				iMinute:=BYTE_TO_INT(recBuf[9]-48)*10+BYTE_TO_INT(recBuf[10]-48);
				iSecond:=BYTE_TO_INT(recBuf[11]-48)*10+BYTE_TO_INT(recBuf[12]-48);
			END_IF
				// 计算时间戳		
				strDateTimeNow := CONCAT(STR1 := 'DT#', STR2 := INT_TO_STRING(iYear));
				strDateTimeNow := CONCAT(STR1 := strDateTimeNow, STR2 := '-');
				strDateTimeNow := CONCAT(STR1 := strDateTimeNow, STR2 := INT_TO_STRING(iMonth));
				strDateTimeNow := CONCAT(STR1 := strDateTimeNow, STR2 := '-');
				strDateTimeNow := CONCAT(STR1 := strDateTimeNow, STR2 := INT_TO_STRING(iDay));
				strDateTimeNow := CONCAT(STR1 := strDateTimeNow, STR2 := '-');
				strDateTimeNow := CONCAT(STR1 := strDateTimeNow, STR2 := INT_TO_STRING(iHour));
				strDateTimeNow := CONCAT(STR1 := strDateTimeNow, STR2 := ':');
				strDateTimeNow := CONCAT(STR1 := strDateTimeNow, STR2 := INT_TO_STRING(iMinute));
				strDateTimeNow := CONCAT(STR1 := strDateTimeNow, STR2 := ':');
				strDateTimeNow := CONCAT(STR1 := strDateTimeNow, STR2 := INT_TO_STRING(iSecond));
				gnssTimestamp := DT_TO_ULINT(TO_DT(strDateTimeNow)) * 1000;
				GVL.stGNSS_Timestap := gnssTimestamp;
			//END_IF
		END_IF
					


(*	IF recsize>0 THEN					//如果接收到串口数据
		
		com_write(						//串口发送功能块
		EN_IN:=TRUE,					//串口发送功能块使能，发送机制：当使能为TRUE时，PLC程序每周期运行到此处就执行一次发送
		bPort:=mPort,					//串口端口号设定
		p_bTxdata:=ADR(recbuf),			//将接收存放到数组中的数据发送出去******若发送其它数据，自建另一数组用于存放发送数据即可
		uiTxsize:=recsize,				//发送长度为接收到的数据长度******若发送其它长度，自行填写所需长度即可
		EN_OUT=>m_out,					//串口发送功能块执行完成标志位
		uierror=>m_uierror);			//串口发送功能块执行错误信息
			
	END_IF
*)	
END_IF

END_PROGRAM

// Device/Application/PID_1
FUNCTION_BLOCK PID_1
VAR_INPUT
    rTarget : REAL;       (* 设定值 *)
    rFeedback : REAL;       (* 反馈值 *)
	rPosLimPositive:LREAL;//位置正限位
	rPosLimNegative:LREAL;//位置反限位
	rKp:REAL;     //比例增益
	rKi:REAL;     //积分增益
	rKd:REAL;     //微分增益
	iThreshold:INT;//积分项开启的位置阈值
	bPIDEnable:BOOL:=TRUE;//PID使能
	rVelLim:LREAL;//速度限制
END_VAR
VAR_OUTPUT
    rPIDOutput : LREAL:=0;         //带方向的输出速度

END_VAR
VAR
	//rPIDOutPut: REAL:=0.0;
	rLastError: LREAL:=0.0;(*上一次误差*)
	rErrorNow:LREAL:=0.0;(*当前误差*)
    rIntegralNew : LREAL := 0.0; (* 积分项 *)
    rDerivativeNew : LREAL := 0.0; (* 微分项 *)
	rDelta: LREAL;(*增量*)
	rProportionNew: LREAL;
	
	//iAzPIDEnable: INT;
END_VAR


IF (bPIDEnable>0) THEN //如果PID使能
	IF rTarget=rFeedback THEN
		rPIDOutput:=0;	
	ELSE
	
		rErrorNow:=rTarget-rFeedback;//计算当前误差 en
		rProportionNew:=rErrorNow;//比例项
		//积分项
		IF rFeedback>rPosLimNegative AND rFeedback<rPosLimPositive THEN //若在软限位之内，工作时开启积分项
			IF (ABS(rTarget-rFeedback)<iThreshold OR iThreshold = -1) THEN//位置差小于积分阈值开始积分，或者设置阈值为-1，不启用这个控制
				rIntegralNew:= rIntegralNew+rErrorNow; //积分项
			ELSE
				rIntegralNew:=0;
			END_IF;
		ELSE //不在软限位范围内,则积分项为0
			rIntegralNew:=0;
		END_IF

		//PID输出
		rPIDOutPut:=rKp*rProportionNew+rKi*rIntegralNew;


		//PID限速
		
			IF rPIDOutput<(-rVelLim) THEN
				rPIDOutput:=-rVelLim;
			ELSIF rPIDOutput>rVelLim THEN
				rPIDOutput:=rVelLim;
			END_IF
		
		
		IF rFeedback>rPosLimPositive AND rPIDOutput>0 THEN 
			rPIDOutput:=0;
		END_IF
		IF rFeedback<rPosLimNegative AND rPIDOutput<0 THEN
			rPIDOutput:=0;
		END_IF
		
		rLastError:=rErrorNow;//将当前误差赋值给上一次误差
		
	END_IF
ELSE//非使能清零PID各项
	rProportionNew:=0.0;
	rIntegralNew:=0.0;
	rPIDOutput:=0.0;
END_IF

END_FUNCTION_BLOCK

// Device/Application/GetACUTime
PROGRAM GetACUTime
VAR
    tp      : TP;           // 脉冲定时器
    toggle  : BOOL := FALSE; // 当前输出状态
    clk     : BOOL := FALSE; // 方波输出
    tick_ms : TIME := T#500MS; // 高电平/低电平持续时间
	Result : RTS_IEC_RESULT;
	stUTC_Timestamp :SYSTIME ;
	
	dRTime:ULINT;//上位机外部时间 单位ns Unix时间戳，起点是1970-1-1 0:0:0
	dModbusTime:ULINT;//Modbus临时外部时间
	iCountRemote:INT; //上位机锁定判断时间常数
	dCountRemote:ULINT;//上位机时间滑动平均常数
	dLastRTime:ULINT;//上位机上一次外部时间 单位ns Unix时间戳，起点是1970-1-1 0:0:0
	iDiffRTime:DINT;//上位机时间差值
	dDelRTime:LINT;
	dMeanDelRTime:LINT;
	rTriger:Standard.R_TRIG;//上升沿触发器
	
	iDiff:DINT;//实际时间差值
	iDiffLocal:DINT;//本地时间差值
	iDiffETime:DINT;//外部时间差值
	ulACUTimeStamp : ULINT;
END_VAR


// 每次TP结束时翻转状态
IF NOT tp.Q THEN
    toggle := NOT toggle;
    tp.IN := TRUE;
    tp.PT := tick_ms;
ELSE
    tp.IN := FALSE;
END_IF

tp();

Result := SysTimeRtcHighResGet(stUTC_Timestamp);
rTriger(CLK:=toggle);
IF rTriger.Q THEN
	dRTime := modbus_slave.UTC_New;
	iDiffRTime:=ULINT_TO_DINT(dRTime-dLastRTime);
	IF ABS(iDiffRTime)>500 THEN //两次PTP时间差如果大于500毫秒,则判断为上位机时间失锁
		iCountRemote:=0;
		dCountRemote:=0;
		GVL.bRemoteTimeLock:=FALSE;
	ELSE//否则判断为上位机时间锁定并累计1分钟
		iCountRemote:=iCountRemote+1;
	END_IF
	
	IF iCountRemote>=20 THEN //累计20s认为时间可用
		iCountRemote:=20;
		dDelRTime := TO_ULINT(stUTC_Timestamp) - (dRTime + 8 * 3600 *1000);
		GVL.bRemoteTimeLock:=TRUE;
		//对外部和本机时间差做1分钟的均值滤波
	END_IF
	//GVL.dRemoteTime:=stUTC_Timestamp*1000000 - dMeanDelRTime;
	dLastRTime:=dRTime;
	(*
	IF GVL.bRemoteTimeLock THEN
		dCountRemote:= dCountRemote + 1;
		IF dCountRemote < 10000 THEN
			dMeanDelRTime := (dMeanDelRTime*(dCountRemote-1) + dDelRTime)/dCountRemote;
		ELSE
			dCountRemote := 10000;
			dMeanDelRTime := (dMeanDelRTime*(dCountRemote-1) + dDelRTime)/dCountRemote; 	
			//iDiff:=ULINT_TO_DINT(Gvl.dPTPCSTTime-dLastCSTtime);
			//dLastCSTtime:=dCSTTime;
		END_IF
	END_IF
	*)
END_IF

ulACUTimeStamp := stUTC_Timestamp - dDelRTime;

END_PROGRAM

// Device/Application/XPTOD_SerialCom
PROGRAM XPTOD_SerialCom
VAR
        com_init:gcan.FB_Com_Init;                      //gcan.FB_Com_Init为串口初始化功能块，可设定串口端口号，串口波特率等参数
        com_read:gcan.FB_Com_Read ;                                //gcan.FB_Com_Read为串口接收功能块，用于通过接收串口发送给PLC的数据
        com_write:gcan.FB_Com_Write ;                        //gcan.FB_Com_Write为串口发送功能块，用于发送串口数据
        m_uiError:UINT;                                                        //用于承接功能块中报错引脚错误信息的变量
        m_out:BOOL;                                                                //用于承接功能块中完成标志引脚数据的变量
        isFirst:BOOL:=TRUE;                                                //用于判断初始化只执行一次的逻辑
        mPort:BYTE;                                                                //程序中用作设定串口端口号
        recSize:UINT;                                                        //接收数据长度，单位：字节
        recBuf:ARRAY[0..239] OF BYTE;                        //用于存放接收到的串口数据的数组
        iYear: INT;                             //年
        iMonth: INT;                            //月
        iDay: INT;                              //日
        iHour: INT;                             //时
        iMinute: INT;                           //分
        iSecond: INT;                           //秒
    bChecksumValid: BOOL := FALSE;                //校验和
        nFrameHeadPos: INT := 0;                //帧头索引          
    nPos        : INT;                      //帧头位置
    nChecksumRx : BYTE := 0;                //和校验
        strDateTimeNow : STRING;
        gnssTimestamp: ULINT;
        gnssTimestamplast:ULINT;
        icount:INT;
END_VAR

////////////////////////////////////////////////////////////////////////////////////////
//串口接收TOD报文解析
//日期：2025/05/15
//版本：V1.1
/////////////////////////////////////////////////////////////////////////////////////////

mPort:=1;                                                                //串口端口号设定，GCAN-PLC-400、GCAN-PLC-510、GCAN-PLC-511，1为232，2为485
                                                                                //GCAN-PLC-324、GCAN-PLC-326，1为第一路485，2为第2路485
IF isFirst THEN
        com_init(                                                        //串口初始化功能块
        EN_IN:=TRUE,                                                //串口初始化功能块使能
        xEnable:=TRUE,                                                //串口功能使能
        bPort:=mPort,                                                //串口端口号设定
        uiBaudrate:=115200,                                        //串口波特率设定
        bParity:=0,                                                        //串口奇偶校验设定，0为无校验，1为奇校验，2为偶检验
        bDatabits:=8,                                                //数据位设定
        bStopbits:=1,                                                //停止位设定
        EN_OUT=>m_out,                                                //串口初始化功能块执行完成标志位
        uiError=>m_uiError);                                //串口初始化功能块执行错误信息
        isfirst:=FALSE;                                                //执行一次初始化后关闭IF的条件使其之后进入ELSE程序段运行

ELSE
        
                com_read(                                                //串口读取功能块
                EN_in:=TRUE,                                        //读取功能块使能，为TRUE执行读取
                bPort:=mPort,                                        //串口端口号设定
                p_brxdata:=ADR(recBuf),                        //读取到的串口数据引脚为指针类型，使用ADR()指向自建数组将数据存放到数组中
                uiMaxsize:=240,                                        //设定最大读取长度
                EN_out=>m_out,                                        //串口读取功能块执行完成标志位******功能块执行完成不代表接收完成********
                uiRecSize=>recSize,                                //串口接收数据长度，单位：字节，大于0时说明接收到数据可用于判断是否接收
                uierror=>m_uierror);                        //串口读取功能块执行错误信息
                // 查找帧头 $X (36, 88)
                FOR nPos := 1 TO 240 DO
                        IF recBuf[nPos] = 36 AND recBuf[nPos + 1] = 88 THEN
                                nFrameHeadPos := nPos;
                                EXIT;
                        END_IF
                END_FOR
                //解析时间日期 
                IF nFrameHeadPos + 26 <= 240 THEN
                        iYear:=BYTE_TO_INT(recBuf[nFrameHeadPos+23]-48)*1000+BYTE_TO_INT(recBuf[nFrameHeadPos+24]-48)*100+BYTE_TO_INT(recBuf[nFrameHeadPos+25]-48)*10+BYTE_TO_INT(recBuf[26]-48);
                        iMonth:=BYTE_TO_INT(recBuf[nFrameHeadPos+20]-48)*10+BYTE_TO_INT(recBuf[nFrameHeadPos+21]-48);
                        iDay:=BYTE_TO_INT(recBuf[nFrameHeadPos+17]-48)*10+BYTE_TO_INT(recBuf[nFrameHeadPos+18]-48);
                        iHour:=BYTE_TO_INT(recBuf[nFrameHeadPos+7]-48)*10+BYTE_TO_INT(recBuf[nFrameHeadPos+8]-48)+8;
                        iMinute:=BYTE_TO_INT(recBuf[nFrameHeadPos+9]-48)*10+BYTE_TO_INT(recBuf[nFrameHeadPos+10]-48);
                        iSecond:=BYTE_TO_INT(recBuf[nFrameHeadPos+11]-48)*10+BYTE_TO_INT(recBuf[nFrameHeadPos+12]-48);
                        // 计算时间戳                
                        
                        strDateTimeNow := CONCAT(STR1 := 'DT#', STR2 := INT_TO_STRING(iYear));
                        strDateTimeNow := CONCAT(STR1 := strDateTimeNow, STR2 := '-');
                        strDateTimeNow := CONCAT(STR1 := strDateTimeNow, STR2 := INT_TO_STRING(iMonth));
                        strDateTimeNow := CONCAT(STR1 := strDateTimeNow, STR2 := '-');
                        strDateTimeNow := CONCAT(STR1 := strDateTimeNow, STR2 := INT_TO_STRING(iDay));
                        strDateTimeNow := CONCAT(STR1 := strDateTimeNow, STR2 := '-');
                        strDateTimeNow := CONCAT(STR1 := strDateTimeNow, STR2 := INT_TO_STRING(iHour));
                        strDateTimeNow := CONCAT(STR1 := strDateTimeNow, STR2 := ':');
                        strDateTimeNow := CONCAT(STR1 := strDateTimeNow, STR2 := INT_TO_STRING(iMinute));
                        strDateTimeNow := CONCAT(STR1 := strDateTimeNow, STR2 := ':');
                        strDateTimeNow := CONCAT(STR1 := strDateTimeNow, STR2 := INT_TO_STRING(iSecond));
                        
                        gnssTimestamplast:=gnssTimestamp;
                        gnssTimestamp := DT_TO_ULINT(TO_DT(strDateTimeNow)) * 1000;
                        GVL.stGNSS_Timestap := gnssTimestamp;                        
                END_IF
                
                IF gnssTimestamplast<>gnssTimestamp THEN
                        icount:=0;
                ELSE
                        icount:=icount+1;
                END_IF        
END_IF

END_PROGRAM

// Device/Application/GPRMC_1_1
PROGRAM GPRMC_1_1
VAR
        com_init:gcan.FB_Com_Init;                      //gcan.FB_Com_Init为串口初始化功能块，可设定串口端口号，串口波特率等参数
        com_read:gcan.FB_Com_Read ;                                //gcan.FB_Com_Read为串口接收功能块，用于通过接收串口发送给PLC的数据
        com_write:gcan.FB_Com_Write ;                        //gcan.FB_Com_Write为串口发送功能块，用于发送串口数据
        m_uiError:UINT;                                                        //用于承接功能块中报错引脚错误信息的变量
        m_out:BOOL;                                                                //用于承接功能块中完成标志引脚数据的变量
        isFirst:BOOL:=TRUE;                                                //用于判断初始化只执行一次的逻辑
        mPort:BYTE;                                                                //程序中用作设定串口端口号
        recSize:UINT;                                                        //接收数据长度，单位：字节
        recBuf:ARRAY[0..120] OF BYTE;                        //用于存放接收到的串口数据的数组
        iYear: INT;                             //年
        iMonth: INT;                            //月
        iDay: INT;                              //日
        iHour: INT;                             //时
        iMinute: INT;                           //分
        iSecond: INT;                           //秒
    bChecksumValid: BOOL := FALSE;                //校验和
        nFrameHeadPos: INT := 0;                //帧头索引          
    nPos        : INT;                      //帧头位置
    nChecksumRx : BYTE := 0;                //和校验
        strDateTimeNow : STRING;
        gnssTimestamp: ULINT;
        gnssTimestamplast:ULINT;
        icount:INT;
END_VAR

////////////////////////////////////////////////////////////////////////////////////////
//串口接收TOD报文解析
//日期：2025/05/15
//版本：V1.1
/////////////////////////////////////////////////////////////////////////////////////////

mPort:=1;                                                                //串口端口号设定，GCAN-PLC-400、GCAN-PLC-510、GCAN-PLC-511，1为232，2为485
                                                                                //GCAN-PLC-324、GCAN-PLC-326，1为第一路485，2为第2路485
IF isFirst THEN
        com_init(                                                        //串口初始化功能块
        EN_IN:=TRUE,                                                //串口初始化功能块使能
        xEnable:=TRUE,                                                //串口功能使能
        bPort:=mPort,                                                //串口端口号设定
        uiBaudrate:=115200,                                        //串口波特率设定
        bParity:=0,                                                        //串口奇偶校验设定，0为无校验，1为奇校验，2为偶检验
        bDatabits:=8,                                                //数据位设定
        bStopbits:=1,                                                //停止位设定
        EN_OUT=>m_out,                                                //串口初始化功能块执行完成标志位
        uiError=>m_uiError);                                //串口初始化功能块执行错误信息
        isfirst:=FALSE;                                                //执行一次初始化后关闭IF的条件使其之后进入ELSE程序段运行

ELSE
        
                com_read(                                                //串口读取功能块
                EN_in:=TRUE,                                        //读取功能块使能，为TRUE执行读取
                bPort:=mPort,                                        //串口端口号设定
                p_brxdata:=ADR(recBuf),                        //读取到的串口数据引脚为指针类型，使用ADR()指向自建数组将数据存放到数组中
                uiMaxsize:=240,                                        //设定最大读取长度
                EN_out=>m_out,                                        //串口读取功能块执行完成标志位******功能块执行完成不代表接收完成********
                uiRecSize=>recSize,                                //串口接收数据长度，单位：字节，大于0时说明接收到数据可用于判断是否接收
                uierror=>m_uierror);                        //串口读取功能块执行错误信息
                // 查找帧头 $X (36, 88)
                FOR nPos := 0 TO 119 DO
                        IF recBuf[nPos] = 36 AND recBuf[nPos + 1] = 88 THEN
                                nFrameHeadPos := nPos;
                                EXIT;
                        END_IF
                END_FOR
                //解析时间日期 
                IF nFrameHeadPos + 26 <= 120 THEN
                        iYear:=BYTE_TO_INT(recBuf[nFrameHeadPos+23]-48)*1000+BYTE_TO_INT(recBuf[nFrameHeadPos+24]-48)*100+BYTE_TO_INT(recBuf[nFrameHeadPos+25]-48)*10+BYTE_TO_INT(recBuf[26]-48);
                        iMonth:=BYTE_TO_INT(recBuf[nFrameHeadPos+20]-48)*10+BYTE_TO_INT(recBuf[nFrameHeadPos+21]-48);
                        iDay:=BYTE_TO_INT(recBuf[nFrameHeadPos+17]-48)*10+BYTE_TO_INT(recBuf[nFrameHeadPos+18]-48);
                        iHour:=BYTE_TO_INT(recBuf[nFrameHeadPos+7]-48)*10+BYTE_TO_INT(recBuf[nFrameHeadPos+8]-48)+8;
                        iMinute:=BYTE_TO_INT(recBuf[nFrameHeadPos+9]-48)*10+BYTE_TO_INT(recBuf[nFrameHeadPos+10]-48);
                        iSecond:=BYTE_TO_INT(recBuf[nFrameHeadPos+11]-48)*10+BYTE_TO_INT(recBuf[nFrameHeadPos+12]-48);
                        // 计算时间戳                
                        
                        strDateTimeNow := CONCAT(STR1 := 'DT#', STR2 := INT_TO_STRING(iYear));
                        strDateTimeNow := CONCAT(STR1 := strDateTimeNow, STR2 := '-');
                        strDateTimeNow := CONCAT(STR1 := strDateTimeNow, STR2 := INT_TO_STRING(iMonth));
                        strDateTimeNow := CONCAT(STR1 := strDateTimeNow, STR2 := '-');
                        strDateTimeNow := CONCAT(STR1 := strDateTimeNow, STR2 := INT_TO_STRING(iDay));
                        strDateTimeNow := CONCAT(STR1 := strDateTimeNow, STR2 := '-');
                        strDateTimeNow := CONCAT(STR1 := strDateTimeNow, STR2 := INT_TO_STRING(iHour));
                        strDateTimeNow := CONCAT(STR1 := strDateTimeNow, STR2 := ':');
                        strDateTimeNow := CONCAT(STR1 := strDateTimeNow, STR2 := INT_TO_STRING(iMinute));
                        strDateTimeNow := CONCAT(STR1 := strDateTimeNow, STR2 := ':');
                        strDateTimeNow := CONCAT(STR1 := strDateTimeNow, STR2 := INT_TO_STRING(iSecond));
                        
                        gnssTimestamplast:=gnssTimestamp;
                        gnssTimestamp := DT_TO_ULINT(TO_DT(strDateTimeNow)) * 1000;
                        GVL.stGNSS_Timestap := gnssTimestamp;                        
                END_IF
                
                IF gnssTimestamplast<>gnssTimestamp THEN
                        icount:=0;
                ELSE
                        icount:=icount+1;
                END_IF        
END_IF

END_PROGRAM

// Device/Application/插值模块/LinearInter
FUNCTION_BLOCK LinearInter
VAR_INPUT
	tLastTime:ULINT;//上一时间
	rLastPos:REAL;//上一时间位置
	
	tCurTime:ULINT;//当前时间
	rCurPos:REAL;//当前时间位置
	
	tTargetTime:ULINT;//目标时间
END_VAR
VAR_OUTPUT
	rTargetpos:REAL;//目标时间位置
END_VAR
VAR
	iDelCurLastTime:LREAL:=1.0;//	当前与上一个时间差
	iDelTarCurTime:LREAL:=1.0;//目标与当前时间差
	rK:REAL;//方位斜率
END_VAR

//tLastTime:=tLastTime/1000000;
//tCurTime:=tCurTime/1000000;
//tTargetTime:=tTargetTime/1000000;
iDelTarCurTime:=ULINT_TO_LREAL(tTargetTime)-ULINT_TO_LREAL(tCurTime); //x1-x
IF (tCurTime-tLastTime)<>0 THEN
	iDelCurLastTime:=ULINT_TO_LREAL(tCurTime)-ULINT_TO_LREAL(tLastTime);  //x-x0
ELSE
	iDelCurLastTime:=1.0;
END_IF

IF iDelTarCurTime<>0 THEN
	rK:=(rCurPos-rLastPos)/(iDelCurLastTime);
ELSE
	rK:=0;
END_IF
rTargetpos:=rCurPos+rK*iDelTarCurTime;  //y1 + ((y1-y0)/(x1-x0))*(x-x1)

END_FUNCTION_BLOCK

// Device/Application/插值模块/threesimple2
FUNCTION_BLOCK threesimple2
VAR_INPUT
	aUTC_TIME:ARRAY [1..5] OF ULINT;  //用于三次样条插值的数据
	aPosCmd :ARRAY [1..5] OF LREAL;//用于三次样条插值的数据
	
	y0:REAL;
	yn:REAL;//y0,yn表示的是S''(x0)=f''(x0)=y0，S''(xn)=f''(xn)=yn,自然边界即条件值为0
	xt:REAL;//所求目标位置
END_VAR
VAR_OUTPUT
	sout:REAL;
	nout:INT;
END_VAR
VAR
	Three:three2;
	X:ARRAY [1..5] OF LREAL;
	Y:ARRAY [1..5] OF LREAL;
	M :ARRAY [1..5] OF LREAL;
	A: ARRAY [1..5,1..5] OF LREAL;
	D: ARRAY[1..3,1..3] OF LREAL;
	g: ARRAY [1..3] OF LREAL;
	h:ARRAY [1..4] OF LREAL;
	
	n:INT:=5;
	
	p1: ARRAY [1..4] OF REAL;
	p2:ARRAY [1..4] OF REAL;
	p3:ARRAY [1..4] OF REAL;
	p4:ARRAY [1..4] OF REAL;
	i:INT;
	
END_VAR

FOR i:=1 TO 5 DO
	X[i]:=ULINT_TO_LREAL(aUTC_TIME[i]);
	Y[i]:=aPosCmd[i];
END_FOR


Three(X:=X,Y:=Y,y0:=y0,yn:=yn,D=>D,h=>h,A=>A,g=>g,M=>M);

FOR i:=1 TO (n-1) DO
	p1[i]:=M[i]*(X[i+1]-xt)*(X[i+1]-xt)*(X[i+1]-xt)/(6*h[i]);
	p2[i]:=M[i+1]*(xt-X[i])*(xt-X[i])*(xt-X[i])/(6*h[i]);
	p3[i]:=(A[i,1]-M[i]/6*(h[i])*(h[i]))*(X[i+1]-xt)/h[i];
	p4[i]:=(A[i+1,1]-M[i+1]/6*(h[i])*(h[i]))*(xt-X[i])/h[i];
	
	
END_FOR


FOR i:=1 TO (n-1) DO
	IF (xt<=X[i+1])AND (xt>=X[i]) THEN
		nout:=i;
		sout:=p1[nout]+p2[nout]+p3[nout]+p4[nout]; 
	ELSIF xt>X[5] THEN
		nout:=4;
	ELSIF xt<X[1]THEN
		nout:=1;
	END_IF
END_FOR


//要不要判断插值模块是否有效？
sout:=p1[nout]+p2[nout]+p3[nout]+p4[nout]; 
(*
IF xt>X[5] THEN
	nout:=4;
	sout:=p1[nout]+p2[nout]+p3[nout]+p4[nout]; 
ELSIF xt<X[1] THEN
	nout:=1;
	sout:=p1[nout]+p2[nout]+p3[nout]+p4[nout]; 
END_IF
*)

END_FUNCTION_BLOCK

// Device/Application/插值模块/InterDataProcess
FUNCTION_BLOCK InterDataProcess
VAR_INPUT
	ulRealTime: ULINT;//实际时间 单位纳秒
	//aOrbitTime: ARRAY [1..5] OF ULINT;//轨道时间数组
	Arr: ARRAY [1..5] OF ULINT:=[9,0,1,5,4]; // 创建一个包含5个整数的数组 轨道时间数组  起点 1970-01-01 0:00:00 单位纳秒
    
END_VAR
VAR_OUTPUT
	MaxVal, MinVal: ULINT;   // 定义最大值、最小值和循环计数器变量
    MaxIndex, MinIndex: INT; // 定义最大值和最小值的索引
	ulInterRealTime : ULINT;//插值使用的时间
END_VAR
VAR
	i,j: INT;
END_VAR

//该功能块查找到轨道时间数组内最大最小值以及索引位置
//找出最大最小值
MaxVal := 0; // 初始化最大值
MinVal := 0; // 初始化最小值
MaxIndex := 0; // 初始化最大值的索引
MinIndex := 0; // 初始化最小值的索引

FOR i := 1 TO 5 DO
    IF Arr[i] <> 0 THEN
        IF MaxVal = 0 THEN
            MaxVal := Arr[i];
            MaxIndex := i;
        ELSIF Arr[i] > MaxVal THEN
            MaxVal := Arr[i];
            MaxIndex := i;
        END_IF

        IF MinVal = 0 THEN
            MinVal := Arr[i];
            MinIndex := i;
        ELSIF Arr[i] < MinVal THEN
            MinVal := Arr[i];
            MinIndex := i;
        END_IF
    END_IF
END_FOR

// MaxVal 和 MinVal 包含了最大值和最小值，不考虑值为0的元素
// MaxIndex 和 MinIndex 包含了最大值和最小值的索引


//当前时间和最大最小比较 
IF ulRealTime<MinVal*1000000 THEN //小于插值范围 取最小时间
	//
	ulInterRealTime:=MinVal*1000000; //应该修改插值位置 而不是时间
ELSIF ulRealTime>MaxVal*1000000THEN //大于插值范围 取最大时间
	//
	ulInterRealTime:=MaxVal*1000000;//应该修改插值位置 而不是时间
ELSE
	//如果内部有0 则不插值选取最新的数据
	FOR j:=1 TO 5 DO
		IF (Arr[i]=0) AND (j<5) THEN
			ulInterRealTime:=Arr[5];//应该修改插值位置 而不是时间
			MaxIndex:=5;
			EXIT;
		ELSIF (Arr[i]=0) AND (j=5) THEN
			//没有输入数据 需要报错吗？
		END_IF
	END_FOR
	//
END_IF

END_FUNCTION_BLOCK

// /ElCtrl
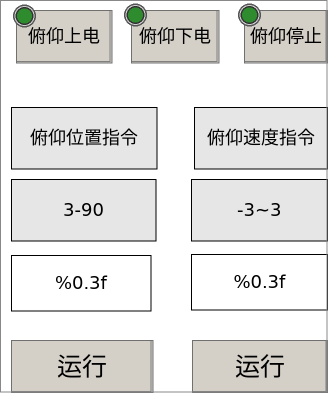
VISUALIZATION ElCtrl  // 328x393
    Button (131,10 88x53), "俯仰下电"
        OnMouseClick: execute { GVL.Axis1Local.iMode:=0; }
    Button (16,10 96x53), "俯仰上电"
        OnMouseClick: execute { GVL.Axis1Local.iMode:=1; }
    Lamp1 (6,3 37x26), variable: GVL.Axis1Status.bServo_Enable, style: Lamp-Lamp1-Green
    Lamp1 (117,2 37x26), variable: NOT(GVL.Axis1Status.bServo_Enable), style: Lamp-Lamp1-Green
    Button (244,10 84x53), "俯仰停止"
        OnMouseClick: execute { GVL.Axis1Local.iMode:=7; }
    Lamp1 (231,2 37x26), variable: NOT(GVL.Axis1Status.Moving), style: Lamp-Lamp1-Green
    Rectangle (11,107 146x62), "俯仰位置指令"
    Rectangle (11,255 140x56), "%0.3f", text variable: ElV.rPosCmd
        OnMouseClick: write the text variable via Default, min 3, max 90
    Button (11,340 142x53), "运行"
        OnMouseClick: execute {
            GVL.Axis1Local.rPosCmd:=GVL.ElV.rPosCmd+90;
            GVL.Axis1Local.iMode:=4;
            GVL.Axis1Local.bPIDEnable:=TRUE;
        }
    Rectangle (194,107 134x62), "俯仰速度指令"
    Rectangle (191,254 137x56), "%0.3f", text variable: ElV.rVelCmd
        OnMouseClick: write the text variable via Default, min -10, max 10
    Button (192,340 136x53), "运行"
        OnMouseClick: execute { GVL.Axis1Local.rVelCmd:=GVL.ElV.rVelCmd; GVL.Axis1Local.iMode:=3; }
    Rectangle (11,179 145x62), "3-90"
    Rectangle (191,179 137x62), "-3~3"
END_VISUALIZATION

// Device/Application/可视化/Visualization
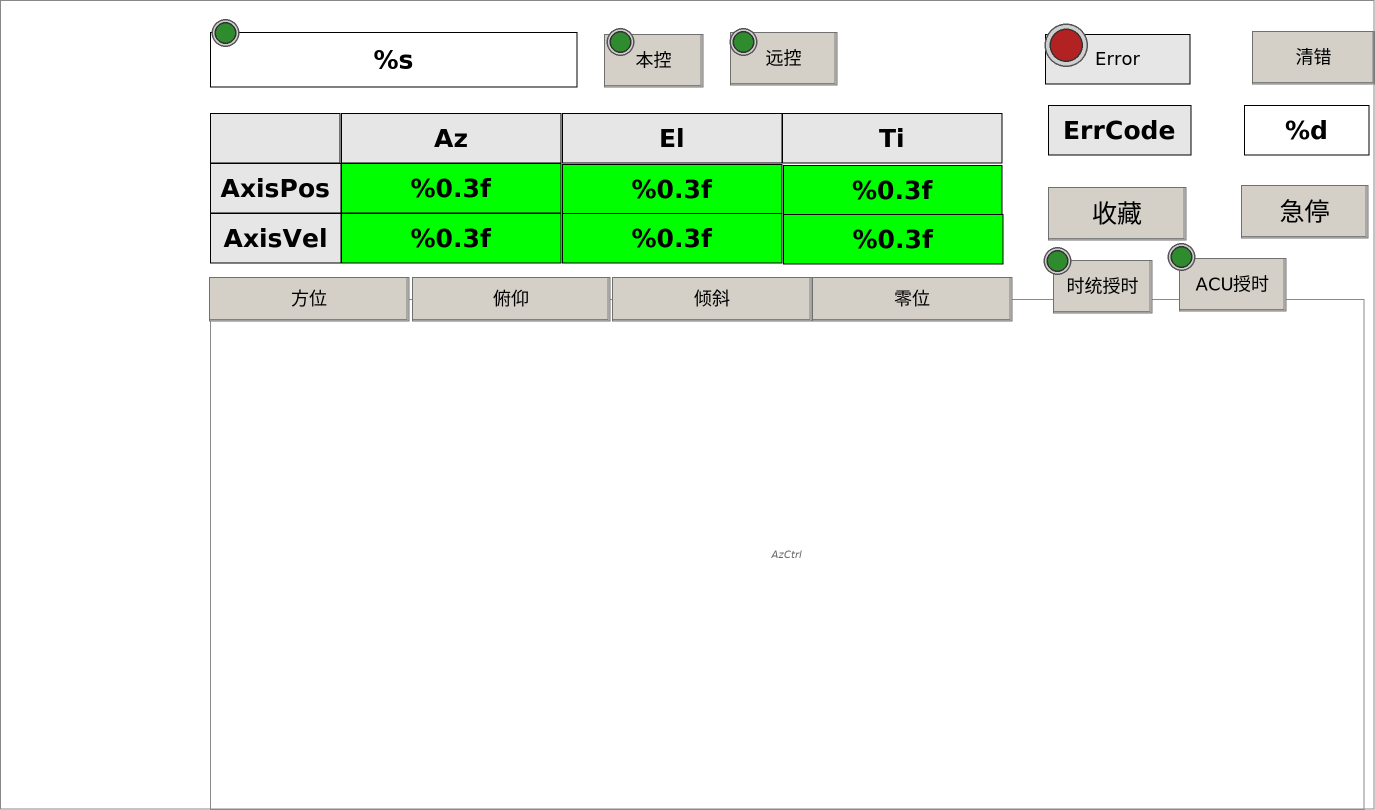
VISUALIZATION Visualization  // 1375x810
    Rectangle (210,32 367x55), "%s", text variable: RealTimePosCal.dtReal
    Button (604,34 99x53), "本控"
        OnMouseClick: execute { GVL.bLocalCtrl:=TRUE; }
    Button (730,32 107x53), "远控"
        OnMouseClick: execute { GVL.bLocalCtrl:=FALSE; }
    Lamp1 (596,26 49x32), variable: GVL.bLocalCtrl, style: Lamp-Lamp1-Green
    Lamp1 (721,26 45x32), variable: NOT(GVL.bLocalCtrl), style: Lamp-Lamp1-Green
    Rectangle (341,113 220x50), "Az"
    Rectangle (562,113 220x50), "El"
    Rectangle (210,163 131x50), "AxisPos"
    Rectangle (341,163 220x50), "%0.3f", text variable: GVL.rFctPosReal_2*(-1)
    Rectangle (562,164 220x50), "%0.3f", text variable: GVL.rFctPosReal_1-90
    Rectangle (210,113 130x50)
    Rectangle (210,213 131x50), "AxisVel"
    Rectangle (341,213 220x50), "%0.3f", text variable: GVL.rFctVelReal_2*(-1)
    Rectangle (562,213 220x50), "%0.3f", text variable: GVL.rFctVelReal_1
    Lamp1 (203,17 45x32), variable: TimeCase.Triger, style: Lamp-Lamp1-Green
    Rectangle (1045,34 145x50), "Error"
    Lamp1 (1026,20 80x50), variable: Az_ctrl_1.bVisError, style: Lamp-Lamp1-Red
    Button (1048,187 138x53), "收藏"
        OnMouseClick: execute {
            GVL.Axis1Local.rPosCmd:=180;
            GVL.Axis1Local.iMode:=4;
            GVL.Axis1Local.bPIDEnable:=TRUE;
            GVL.Axis2Local.rPosCmd:=0;
            GVL.Axis2Local.iMode:=4;
            GVL.Axis2Local.bPIDEnable:=TRUE;
            GVL.Axis3Local.rPosCmd:=0;
            GVL.Axis3Local.iMode:=4;
            GVL.Axis3Local.bPIDEnable:=TRUE;
        }
    Button (1241,185 127x53), "急停"
        OnMouseClick: execute {
            GVL.Axis1Local.iMode:=0;
            GVL.Axis2Local.iMode:=0;
            GVL.Axis3Local.iMode:=0;
        }
    Rectangle (1048,105 143x50), "ErrCode"
    Rectangle (1244,105 125x50), "%d", text variable: GVL.Error_code
    Button (1252,31 123x53), "清错"
        OnMouseClick: execute { GVL.bError_Reset:=TRUE; }
    Rectangle (782,113 220x50), "Ti"
    Rectangle (783,165 219x50), "%0.3f", text variable: GVL.rFctPosReal_3*(-1)
    Rectangle (783,214 220x50), "%0.3f", text variable: GVL.rFctVelReal_3*(-1)
    TabControl (210,299 1154x511), frame switch variable: GVL.iVisualSwitch
        shows AzCtrl()
        shows ElCtrl()
        shows TlCtrl()
        shows north()
        shows IOtest()
        shows IOState()
    Button (209,277 200x44), "方位", input disabled if: GVL.bAzVisable
        OnMouseClick: execute {
            GVL.bAzVisable:=TRUE;
            GVL.bElVisable:=FALSE;
            GVL.bTlVisable:=FALSE;
            GVL.bLocalAutoTrackVis:=FALSE;
            GVL.iVisualSwitch:=0;
        }
    Button (412,277 198x44), "俯仰", input disabled if: GVL.bElVisable
        OnMouseClick: execute {
            GVL.bAzVisable:=FALSE;
            GVL.bElVisable:=TRUE;
            GVL.bTlVisable:=FALSE;
            GVL.bLocalAutoTrackVis:=FALSE;
            GVL.iVisualSwitch:=1;
        }
    Button (612,277 200x44), "倾斜", input disabled if: GVL.bTlVisable
        OnMouseClick: execute {
            GVL.bAzVisable:=FALSE;
            GVL.bElVisable:=FALSE;
            GVL.bTlVisable:=TRUE;
            GVL.bLocalAutoTrackVis:=FALSE;
            GVL.iVisualSwitch:=2;
        }
    Button (812,277 200x44), "零位", input disabled if: GVL.bLocalAutoTrackVis
        OnMouseClick: execute {
            GVL.bAzVisable:=FALSE;
            GVL.bElVisable:=FALSE;
            GVL.bTlVisable:=FALSE;
            GVL.bLocalAutoTrackVis:=TRUE;
            GVL.iVisualSwitch:=3;
        }
    Button (1053,260 99x53), "时统授时"
        OnMouseClick: execute { GVL.bTimeSwich := FALSE; }
    Button (1179,258 107x53), "ACU授时"
        OnMouseClick: execute { GVL.bTimeSwich := TRUE; }
    Lamp1 (1033,245 49x32), variable: NOT(GVL.bTimeSwich), style: Lamp-Lamp1-Green
    Lamp1 (1159,241 45x32), variable: GVL.bTimeSwich, style: Lamp-Lamp1-Green
END_VISUALIZATION

// Device/Application/可视化/ElCtrl
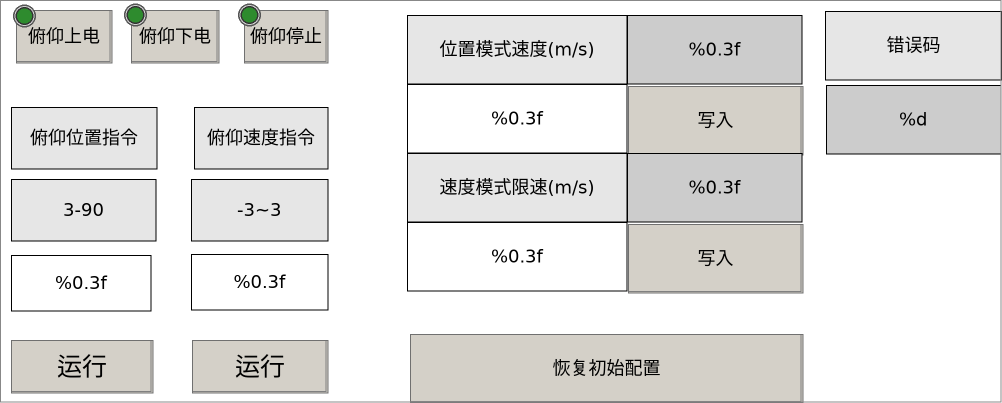
VISUALIZATION ElCtrl  // 1002x403
    Button (131,10 88x53), "俯仰下电"
        OnMouseClick: execute { GVL.Axis1Local.iMode:=0; }
    Button (16,10 96x53), "俯仰上电"
        OnMouseClick: execute { GVL.Axis1Local.iMode:=1; }
    Lamp1 (6,3 37x26), variable: GVL.Axis1Status.bServo_Enable, style: Lamp-Lamp1-Green
    Lamp1 (117,2 37x26), variable: NOT(GVL.Axis1Status.bServo_Enable), style: Lamp-Lamp1-Green
    Button (244,10 84x53), "俯仰停止"
        OnMouseClick: execute { GVL.Axis1Local.iMode:=7; }
    Lamp1 (231,2 37x26), variable: NOT(GVL.Axis1Status.Moving), style: Lamp-Lamp1-Green
    Rectangle (11,107 146x62), "俯仰位置指令"
    Rectangle (11,255 140x56), "%0.3f", text variable: ElV.rPosCmd
        OnMouseClick: write the text variable via Default, min 0, max 90
    Button (11,340 142x53), "运行"
        OnMouseClick: execute {
            GVL.Axis1Local.rPosCmd:=GVL.ElV.rPosCmd+90;
            GVL.Axis1Local.iMode:=4;
            GVL.Axis1Local.bPIDEnable:=TRUE;
        }
    Rectangle (194,107 134x62), "俯仰速度指令"
    Rectangle (191,254 137x56), "%0.3f", text variable: ElV.rVelCmd
        OnMouseClick: write the text variable via Default, min -13, max 13
    Button (192,340 136x53), "运行"
        OnMouseClick: execute { GVL.Axis1Local.rVelCmd:=GVL.ElV.rVelCmd; GVL.Axis1Local.iMode:=3; }
    Rectangle (11,179 145x62), "3-90"
    Rectangle (191,179 137x62), "-3~3"
    Rectangle (627,15 175x69), "%0.3f", text variable: Axis1Local.Pos_Vel
    Rectangle (407,15 220x69), "位置模式速度(m/s)"
    Rectangle (407,84 220x69), "%0.3f", text variable: ElV.Pos_Vel
        OnMouseClick: write the text variable via Edit, min -15.5, max 15.5
    Button (628,86 175x69), "写入"
        OnMouseClick: execute { Axis1Local.Pos_Vel:=ElV.Pos_Vel; }
    Rectangle (627,153 175x69), "%0.3f", text variable: Axis1Local.rVel_Limit
    Rectangle (407,153 220x69), "速度模式限速(m/s)"
    Rectangle (407,222 220x69), "%0.3f", text variable: ElV.rVel_Limit
        OnMouseClick: write the text variable via Edit, min 2, max 11
    Button (628,224 175x69), "写入"
        OnMouseClick: execute { Axis1Local.rVel_Limit:=ElV.rVel_Limit; }
    Button (410,334 393x69), "恢复初始配置"
        OnMouseClick: execute { Axis1Local.rVel_Limit:=3; Axis1Local.Pos_Vel:=4; }
    Rectangle (826,85 175x69), "%d", text variable: GVL.eElErrorcode
    Rectangle (825,11 177x69), "错误码"
END_VISUALIZATION

// Device/Application/可视化/AzCtrl
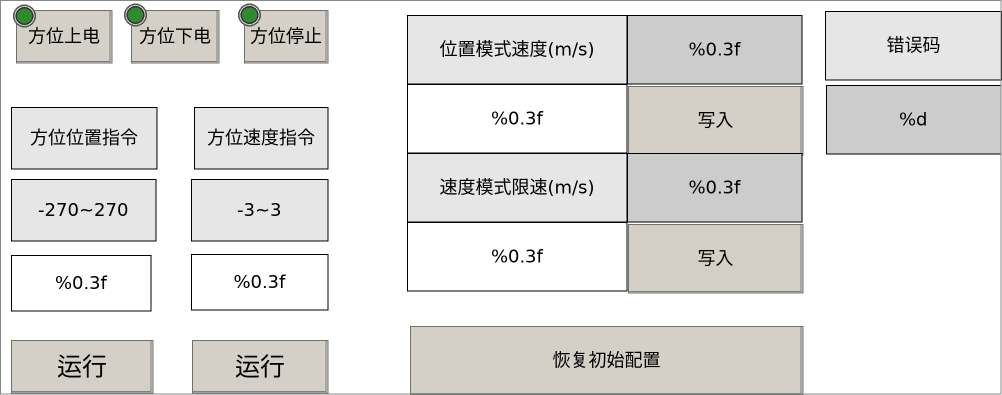
VISUALIZATION AzCtrl  // 1002x395
    Button (131,10 88x53), "方位下电"
        OnMouseClick: execute { GVL.Axis2Local.iMode:=0; }
    Button (16,10 96x53), "方位上电"
        OnMouseClick: execute { GVL.Axis2Local.iMode:=1; }
    Lamp1 (6,3 37x26), variable: GVL.Axis2Status.bServo_Enable, style: Lamp-Lamp1-Green
    Lamp1 (117,2 37x26), variable: NOT(GVL.Axis2Status.bServo_Enable), style: Lamp-Lamp1-Green
    Button (244,10 84x53), "方位停止"
        OnMouseClick: execute { GVL.Axis2Local.iMode:=7; }
    Lamp1 (231,2 37x26), variable: NOT(GVL.Axis2Status.Moving), style: Lamp-Lamp1-Green
    Rectangle (11,107 146x62), "方位位置指令"
    Rectangle (11,255 140x56), "%0.3f", text variable: AzV.rPosCmd
        OnMouseClick: write the text variable via Default, min -270, max 270
    Button (11,340 142x53), "运行"
        OnMouseClick: execute {
            GVL.Axis2Local.rPosCmd:=-GVL.AzV.rPosCmd;
            GVL.Axis2Local.iMode:=4;
            GVL.Axis2Local.bPIDEnable:=TRUE;
        }
    Rectangle (194,107 134x62), "方位速度指令"
    Rectangle (191,254 137x56), "%0.3f", text variable: AzV.rVelCmd
        OnMouseClick: write the text variable via Default, min -20, max 20
    Button (192,340 136x53), "运行"
        OnMouseClick: execute { GVL.Axis2Local.rVelCmd:=GVL.AzV.rVelCmd*(-1); GVL.Axis2Local.iMode:=3; }
    Rectangle (11,179 145x62), "-270~270"
    Rectangle (191,179 137x62), "-3~3"
    Rectangle (627,15 175x69), "%0.3f", text variable: Axis2Local.Pos_Vel
    Rectangle (407,15 220x69), "位置模式速度(m/s)"
    Rectangle (407,84 220x69), "%0.3f", text variable: AzV.Pos_Vel
        OnMouseClick: write the text variable via Edit, min -15.5, max 15.5
    Button (628,86 175x69), "写入"
        OnMouseClick: execute { Axis2Local.Pos_Vel:=AzV.Pos_Vel; }
    Rectangle (627,153 175x69), "%0.3f", text variable: Axis2Local.rVel_Limit
    Rectangle (407,153 220x69), "速度模式限速(m/s)"
    Rectangle (407,222 220x69), "%0.3f", text variable: AzV.rVel_Limit
        OnMouseClick: write the text variable via Edit, min 2, max 15.5
    Button (628,224 175x69), "写入"
        OnMouseClick: execute { Axis2Local.rVel_Limit:=AzV.rVel_Limit; }
    Button (410,326 393x69), "恢复初始配置"
        OnMouseClick: execute { Axis2Local.rVel_Limit:=3; Axis2Local.Pos_Vel:=4; }
    Rectangle (826,85 175x69), "%d", text variable: GVL.eAzErrorcode
    Rectangle (825,11 177x69), "错误码"
END_VISUALIZATION

